  MoveL 1282 to (109.25, -79.9, 66.98) mm, rotated rx 117.25 ry 0 rz -126.43 deg; joints [128.975, -20.959, 32.859, -104.299, 40.472, 146.273, 25, -233.571]
  MoveL 1283 to (108.79, -81.97, 65.21) mm, rotated rx 116.26 ry 0 rz -127.74 deg; joints [128.667, -21.167, 33.266, -104.678, 40.231, 147.678, 25, -232.264]
  MoveL 1284 to (108.14, -83.32, 64.58) mm, rotated rx 116.26 ry 0 rz -127.74 deg; joints [128.686, -21.239, 33.332, -104.662, 40.248, 147.663, 25, -232.264]
  MoveL 1285 to (107.3, -84.35, 64.64) mm, rotated rx 116.25 ry 0 rz -127.85 deg; joints [128.711, -21.281, 33.364, -104.637, 40.269, 147.65, 25, -232.148]
  MoveL 1286 to (106.13, -85.42, 65.16) mm, rotated rx 116.5 ry 0 rz -129 deg; joints [128.756, -21.17, 33.217, -104.574, 40.301, 147.325, 25, -231.004]
  MoveL 1287 to (103.81, -89.56, 63.3) mm, rotated rx 115.13 ry 0 rz -131.76 deg; joints [128.34, -21.422, 33.746, -105.103, 39.98, 149.276, 25, -228.241]
  MoveL 1288 to (103.98, -91.37, 60.39) mm, rotated rx 113.92 ry 0 rz -132.27 deg; joints [127.986, -21.728, 34.311, -105.588, 39.715, 151.018, 25, -227.728]
  Set speed (16.7 mm/s)
  MoveL 1289 to (117.51, -103.67, 68.5) mm, rotated rx 113.92 ry 0 rz -132.27 deg; joints [127.572, -22.198, 34.1, -105.006, 39.145, 150.151, 25, -227.728]
  Set speed (1000.0 mm/s)
  MoveL 1290 to (138.84, -95.44, -29.33) mm, rotated rx 80.82 ry 0 rz -124.03 deg; joints [119.936, -25.445, 49.101, -124.867, 37.461, 205.459, 25, -235.972]
  Set speed (5.0 mm/s)
  MoveL 1291 to (122.47, -84.4, -26.14) mm, rotated rx 80.82 ry 0 rz -124.03 deg; joints [120.661, -24.792, 48.882, -124.547, 38.253, 205.426, 25, -235.972]
  Set speed (16.7 mm/s)
  MoveL 1292 to (121.83, -85.61, -25.22) mm, rotated rx 81.17 ry 0 rz -124.55 deg; joints [120.706, -24.83, 48.75, -124.321, 38.19, 204.807, 25, -235.447]
  MoveL 1293 to (121.51, -86.3, -24.42) mm, rotated rx 81.17 ry 0 rz -124.55 deg; joints [120.731, -24.874, 48.749, -124.248, 38.184, 204.727, 25, -235.447]
  MoveL 1294 to (121.4, -86.6, -23.9) mm, rotated rx 81.37 ry 0 rz -124.67 deg; joints [120.757, -24.895, 48.673, -124.119, 38.149, 204.372, 25, -235.327]
  MoveL 1295 to (121.32, -86.89, -23.19) mm, rotated rx 81.37 ry 0 rz -124.67 deg; joints [120.77, -24.915, 48.66, -124.07, 38.142, 204.317, 25, -235.327]
  MoveL 1296 to (121.66, -86.85, -21.5) mm, rotated rx 81.37 ry 0 rz -124.67 deg; joints [120.783, -24.917, 48.601, -123.991, 38.117, 204.223, 25, -235.327]
  MoveL 1297 to (123.29, -85.43, -17.57) mm, rotated rx 82.88 ry 0 rz -123.88 deg; joints [120.988, -25.05, 48.027, -123.022, 37.884, 201.596, 25, -236.124]
  MoveL 1298 to (123.63, -85.07, -16.92) mm, rotated rx 82.88 ry 0 rz -123.88 deg; joints [120.985, -25.03, 47.991, -123.009, 37.872, 201.577, 25, -236.124]
  MoveL 1299 to (124.64, -83.71, -16.25) mm, rotated rx 82.88 ry 0 rz -123.88 deg; joints [120.955, -24.952, 47.916, -123.043, 37.851, 201.606, 25, -236.124]
  MoveL 1300 to (124.99, -83.19, -16.24) mm, rotated rx 82.88 ry 0 rz -123.63 deg; joints [120.955, -24.952, 47.915, -123.042, 37.85, 201.602, 25, -236.366]
  MoveL 1301 to (125.61, -82.2, -16.51) mm, rotated rx 82.88 ry 0 rz -123.63 deg; joints [120.926, -24.894, 47.886, -123.104, 37.844, 201.666, 25, -236.366]
  MoveL 1302 to (128.29, -77.31, -19.31) mm, rotated rx 81.81 ry 0 rz -121.51 deg; joints [120.778, -24.803, 48.296, -123.794, 38.007, 203.536, 25, -238.495]
  MoveL 1303 to (128.77, -76.11, -20.82) mm, rotated rx 81.81 ry 0 rz -121.51 deg; joints [120.734, -24.729, 48.303, -123.926, 38.018, 203.681, 25, -238.495]
  MoveL 1304 to (128.6, -75.88, -22.52) mm, rotated rx 80.71 ry 0 rz -121.17 deg; joints [120.62, -24.664, 48.706, -124.541, 38.195, 205.508, 25, -238.828]
  MoveL 1305 to (129, -74.93, -23.4) mm, rotated rx 80.37 ry 0 rz -120.78 deg; joints [120.578, -24.627, 48.832, -124.756, 38.256, 206.097, 25, -239.222]
  MoveL 1306 to (129.03, -74.88, -23.37) mm, rotated rx 80.33 ry 0 rz -119.57 deg; joints [120.643, -24.776, 48.942, -124.646, 38.283, 206.031, 25, -240.434]
  MoveL 1307 to (130.64, -72.67, -21.45) mm, rotated rx 81.07 ry 0 rz -118.53 deg; joints [120.735, -24.856, 48.667, -124.175, 38.152, 204.743, 25, -241.473]
  MoveL 1308 to (131.06, -72.02, -21.04) mm, rotated rx 81.13 ry 0 rz -118.38 deg; joints [120.737, -24.845, 48.622, -124.138, 38.134, 204.631, 25, -241.615]
  MoveL 1309 to (133.41, -67.9, -19.93) mm, rotated rx 81.49 ry 0 rz -116.76 deg; joints [120.775, -24.857, 48.464, -123.919, 38.068, 204.011, 25, -243.236]
  MoveL 1310 to (133.8, -67.15, -19.89) mm, rotated rx 81.49 ry 0 rz -116.76 deg; joints [120.757, -24.816, 48.436, -123.951, 38.061, 204.043, 25, -243.236]
  MoveL 1311 to (134.25, -66.19, -20.09) mm, rotated rx 81.47 ry 0 rz -116.6 deg; joints [120.739, -24.783, 48.428, -123.998, 38.062, 204.113, 25, -243.403]
  MoveL 1312 to (135.7, -62.67, -21.57) mm, rotated rx 80.91 ry 0 rz -115.14 deg; joints [120.665, -24.726, 48.641, -124.361, 38.158, 205.101, 25, -244.859]
  MoveL 1313 to (137.15, -59.17, -22.28) mm, rotated rx 80.59 ry 0 rz -113.52 deg; joints [120.636, -24.714, 48.771, -124.54, 38.216, 205.634, 25, -246.485]
  MoveL 1314 to (137.34, -58.68, -22.4) mm, rotated rx 80.55 ry 0 rz -113.37 deg; joints [120.628, -24.703, 48.781, -124.57, 38.222, 205.704, 25, -246.63]
  MoveL 1315 to (138.52, -55.33, -23.62) mm, rotated rx 80.11 ry 0 rz -112.09 deg; joints [120.568, -24.642, 48.941, -124.865, 38.302, 206.49, 25, -247.906]
  MoveL 1316 to (138.88, -54.28, -23.91) mm, rotated rx 79.98 ry 0 rz -111.6 deg; joints [120.556, -24.635, 48.994, -124.94, 38.328, 206.712, 25, -248.398]
  MoveL 1317 to (141.71, -44.3, -27.64) mm, rotated rx 78.56 ry 0 rz -107.69 deg; joints [120.387, -24.444, 49.506, -125.843, 38.61, 209.189, 25, -252.307]
  MoveL 1318 to (141.88, -43.31, -28.3) mm, rotated rx 78.56 ry 0 rz -107.69 deg; joints [120.36, -24.387, 49.493, -125.918, 38.616, 209.27, 25, -252.307]
  MoveL 1319 to (141.91, -42.89, -28.8) mm, rotated rx 78.49 ry 0 rz -107.63 deg; joints [120.344, -24.361, 49.52, -125.988, 38.635, 209.422, 25, -252.372]
  MoveL 1320 to (141.9, -41.96, -30.15) mm, rotated rx 77.64 ry 0 rz -106.92 deg; joints [120.282, -24.295, 49.83, -126.436, 38.812, 210.814, 25, -253.083]
  MoveL 1321 to (142.62, -37.71, -32.31) mm, rotated rx 76.8 ry 0 rz -105.25 deg; joints [120.198, -24.163, 50.124, -126.951, 39.006, 212.263, 25, -254.745]
  MoveL 1322 to (142.69, -36.46, -33.43) mm, rotated rx 76.31 ry 0 rz -105.28 deg; joints [120.125, -24.017, 50.251, -127.3, 39.118, 213.17, 25, -254.72]
  MoveL 1323 to (142.55, -36.21, -34.26) mm, rotated rx 76.05 ry 0 rz -105.29 deg; joints [120.095, -23.958, 50.336, -127.474, 39.184, 213.632, 25, -254.707]
  MoveL 1324 to (141.72, -37.09, -36.6) mm, rotated rx 75.28 ry 0 rz -105.33 deg; joints [120.045, -23.861, 50.642, -127.92, 39.396, 214.954, 25, -254.667]
  MoveL 1325 to (141.78, -34.82, -38.6) mm, rotated rx 74.5 ry 0 rz -104.47 deg; joints [119.981, -23.71, 50.904, -128.385, 39.606, 216.3, 25, -255.53]
  MoveL 1326 to (141.86, -33.98, -39.09) mm, rotated rx 74.35 ry 0 rz -104.18 deg; joints [119.966, -23.674, 50.954, -128.484, 39.649, 216.57, 25, -255.818]
  MoveL 1327 to (141.57, -29.29, -43.66) mm, rotated rx 72.55 ry 0 rz -102.41 deg; joints [119.84, -23.287, 51.539, -129.529, 40.174, 219.654, 25, -257.589]
  MoveL 1328 to (141.21, -28.39, -45.4) mm, rotated rx 72.53 ry 0 rz -102.45 deg; joints [119.81, -23.204, 51.561, -129.658, 40.221, 219.826, 25, -257.553]
  MoveL 1329 to (140.47, -29.16, -47.19) mm, rotated rx 72.51 ry 0 rz -102.48 deg; joints [119.818, -23.207, 51.641, -129.72, 40.276, 219.933, 25, -257.518]
  MoveL 1330 to (139.72, -31.68, -47.77) mm, rotated rx 72.48 ry 0 rz -102.53 deg; joints [119.868, -23.318, 51.748, -129.659, 40.307, 219.911, 25, -257.472]
  MoveL 1331 to (139.19, -35.08, -46.94) mm, rotated rx 72.81 ry 0 rz -103.9 deg; joints [119.889, -23.395, 51.643, -129.47, 40.205, 219.343, 25, -256.101]
  MoveL 1332 to (139.1, -35.47, -46.89) mm, rotated rx 72.85 ry 0 rz -104.14 deg; joints [119.886, -23.392, 51.626, -129.46, 40.194, 219.294, 25, -255.858]
  MoveL 1333 to (138.15, -39.86, -46.17) mm, rotated rx 73.13 ry 0 rz -105.93 deg; joints [119.904, -23.456, 51.534, -129.296, 40.108, 218.805, 25, -254.07]
  MoveL 1334 to (137.98, -40.97, -45.71) mm, rotated rx 73.13 ry 0 rz -105.93 deg; joints [119.931, -23.521, 51.559, -129.229, 40.1, 218.733, 25, -254.07]
  MoveL 1335 to (137.95, -41.43, -45.38) mm, rotated rx 73.26 ry 0 rz -106.11 deg; joints [119.94, -23.551, 51.517, -129.153, 40.061, 218.507, 25, -253.89]
  MoveL 1336 to (137.95, -41.9, -44.95) mm, rotated rx 73.26 ry 0 rz -106.11 deg; joints [119.952, -23.582, 51.52, -129.113, 40.052, 218.463, 25, -253.89]
  MoveL 1337 to (138.12, -44.92, -41.35) mm, rotated rx 75.02 ry 0 rz -107.76 deg; joints [120.047, -23.866, 50.921, -128.179, 39.566, 215.545, 25, -252.236]
  MoveL 1338 to (137.32, -48.01, -40.54) mm, rotated rx 75.35 ry 0 rz -109.02 deg; joints [120.073, -23.928, 50.812, -127.987, 39.479, 214.989, 25, -250.98]
  MoveL 1339 to (137.34, -47.93, -40.55) mm, rotated rx 75.14 ry 0 rz -109.88 deg; joints [120.011, -23.783, 50.791, -128.175, 39.512, 215.397, 25, -250.12]
  MoveL 1340 to (135.25, -51.11, -43.62) mm, rotated rx 73.93 ry 0 rz -111.35 deg; joints [119.917, -23.537, 51.193, -128.891, 39.85, 217.485, 25, -248.653]
  MoveL 1341 to (134.45, -52.71, -44.19) mm, rotated rx 73.93 ry 0 rz -111.35 deg; joints [119.953, -23.617, 51.268, -128.846, 39.872, 217.449, 25, -248.653]
  MoveL 1342 to (134.28, -53.17, -44.17) mm, rotated rx 73.94 ry 0 rz -111.54 deg; joints [119.954, -23.619, 51.264, -128.84, 39.869, 217.429, 25, -248.459]
  MoveL 1343 to (133.34, -55.46, -44.11) mm, rotated rx 73.97 ry 0 rz -112.56 deg; joints [119.954, -23.619, 51.253, -128.83, 39.862, 217.393, 25, -247.435]
  MoveL 1344 to (132.43, -57.68, -44.06) mm, rotated rx 73.98 ry 0 rz -113.52 deg; joints [119.954, -23.623, 51.247, -128.819, 39.856, 217.36, 25, -246.485]
  MoveL 1345 to (132.15, -58.44, -43.91) mm, rotated rx 73.98 ry 0 rz -113.52 deg; joints [119.973, -23.667, 51.27, -128.779, 39.856, 217.319, 25, -246.485]
  MoveL 1346 to (131.99, -58.95, -43.73) mm, rotated rx 74.06 ry 0 rz -113.72 deg; joints [119.978, -23.682, 51.246, -128.736, 39.834, 217.192, 25, -246.275]
  MoveL 1347 to (131, -62.6, -41.54) mm, rotated rx 74.84 ry 0 rz -115.02 deg; joints [120.049, -23.868, 50.997, -128.247, 39.613, 215.819, 25, -244.982]
  MoveL 1348 to (128.38, -67.77, -41.64) mm, rotated rx 74.94 ry 0 rz -117.85 deg; joints [120.024, -23.813, 50.927, -128.26, 39.587, 215.717, 25, -242.151]
  Set speed (16.7 mm/s)
  MoveL 1349 to (145.45, -76.79, -46.84) mm, rotated rx 74.94 ry 0 rz -117.85 deg; joints [119.274, -24.456, 51.216, -128.772, 38.843, 215.939, 25, -242.151]
  Set speed (1000.0 mm/s)
  MoveL 1350 to (145.71, -79, -42.14) mm, rotated rx 75.13 ry 0 rz -117.87 deg; joints [119.357, -24.65, 51.093, -128.369, 38.703, 215.283, 25, -242.133]
  Set speed (5.0 mm/s)
  MoveL 1351 to (128.62, -69.96, -37.01) mm, rotated rx 75.13 ry 0 rz -117.87 deg; joints [120.107, -24.006, 50.807, -127.869, 39.451, 215.072, 25, -242.133]
  Set speed (16.7 mm/s)
  MoveL 1352 to (129.85, -68.52, -35.3) mm, rotated rx 75.8 ry 0 rz -117.14 deg; joints [120.165, -24.128, 50.579, -127.467, 39.279, 213.919, 25, -242.855]
  MoveL 1353 to (129.85, -68.52, -35.32) mm, rotated rx 76.99 ry 0 rz -117 deg; joints [120.26, -24.308, 50.268, -126.882, 39.05, 212.028, 25, -243.001]
  MoveL 1354 to (129.74, -69.29, -34.22) mm, rotated rx 77.8 ry 0 rz -117.78 deg; joints [120.303, -24.361, 49.969, -126.485, 38.871, 210.73, 25, -242.216]
  MoveL 1355 to (129.04, -70.88, -33.63) mm, rotated rx 78.03 ry 0 rz -118.46 deg; joints [120.327, -24.396, 49.888, -126.342, 38.819, 210.329, 25, -241.541]
  MoveL 1356 to (128.8, -71.45, -33.34) mm, rotated rx 78.08 ry 0 rz -118.56 deg; joints [120.341, -24.424, 49.876, -126.287, 38.806, 210.213, 25, -241.44]
  MoveL 1357 to (128.09, -73.34, -31.98) mm, rotated rx 78.67 ry 0 rz -119.48 deg; joints [120.394, -24.489, 49.659, -125.945, 38.679, 209.218, 25, -240.525]
  MoveL 1358 to (127.59, -74.37, -31.59) mm, rotated rx 78.82 ry 0 rz -119.92 deg; joints [120.411, -24.511, 49.604, -125.85, 38.646, 208.953, 25, -240.079]
  MoveL 1359 to (123.08, -82.67, -28.71) mm, rotated rx 79.95 ry 0 rz -123.6 deg; joints [120.537, -24.655, 49.192, -125.145, 38.416, 206.991, 25, -236.396]
  Set speed (16.7 mm/s)
  MoveL 1360 to (139.48, -93.57, -32.2) mm, rotated rx 79.95 ry 0 rz -123.6 deg; joints [119.808, -25.307, 49.422, -125.495, 37.63, 207.055, 25, -236.396]
  Set speed (1000.0 mm/s)
  MoveL 1361 to (86.56, -126.27, -76.23) mm, rotated rx 62.7 ry 0 rz -145.47 deg; joints [118.894, -20.973, 54.737, -135.201, 43.294, 236.447, 25, -214.527]
  Set speed (5.0 mm/s)
  MoveL 1362 to (76.48, -111.63, -67.06) mm, rotated rx 62.7 ry 0 rz -145.47 deg; joints [119.661, -20.42, 54.326, -134.408, 43.847, 235.941, 25, -214.527]
  Set speed (16.7 mm/s)
  MoveL 1363 to (78.17, -110.46, -67.04) mm, rotated rx 62.7 ry 0 rz -144.73 deg; joints [119.655, -20.405, 54.316, -134.418, 43.845, 235.95, 25, -215.272]
  MoveL 1364 to (82.31, -108.27, -65.64) mm, rotated rx 63.33 ry 0 rz -142.43 deg; joints [119.663, -20.682, 54.196, -134.111, 43.574, 234.894, 25, -217.574]
  MoveL 1365 to (83.1, -107.77, -65.47) mm, rotated rx 63.37 ry 0 rz -142.18 deg; joints [119.655, -20.681, 54.173, -134.104, 43.553, 234.839, 25, -217.817]
  MoveL 1366 to (86.56, -105.46, -64.75) mm, rotated rx 63.68 ry 0 rz -140.42 deg; joints [119.653, -20.796, 54.1, -133.964, 43.422, 234.337, 25, -219.58]
  MoveL 1367 to (90.08, -104.34, -61.68) mm, rotated rx 65.21 ry 0 rz -138.47 deg; joints [119.676, -21.383, 53.775, -133.232, 42.807, 231.82, 25, -221.529]
  MoveL 1368 to (92.29, -104.07, -58.82) mm, rotated rx 66.58 ry 0 rz -137.55 deg; joints [119.696, -21.844, 53.439, -132.573, 42.276, 229.569, 25, -222.448]
  MoveL 1369 to (93.65, -103.42, -57.81) mm, rotated rx 66.58 ry 0 rz -137.55 deg; joints [119.665, -21.799, 53.365, -132.585, 42.238, 229.563, 25, -222.448]
  MoveL 1370 to (94.29, -102.92, -57.66) mm, rotated rx 66.61 ry 0 rz -137.46 deg; joints [119.653, -21.778, 53.336, -132.592, 42.225, 229.541, 25, -222.535]
  MoveL 1371 to (95.59, -101.74, -57.6) mm, rotated rx 66.63 ry 0 rz -136.74 deg; joints [119.653, -21.786, 53.329, -132.579, 42.214, 229.497, 25, -223.256]
  MoveL 1372 to (97.07, -100.77, -56.82) mm, rotated rx 67.03 ry 0 rz -135.66 deg; joints [119.68, -21.954, 53.256, -132.353, 42.069, 228.812, 25, -224.345]
  MoveL 1373 to (99.36, -99.94, -54.29) mm, rotated rx 68.34 ry 0 rz -134.37 deg; joints [119.729, -22.38, 52.94, -131.68, 41.604, 226.634, 25, -225.629]
  MoveL 1374 to (99.89, -99.67, -53.81) mm, rotated rx 68.34 ry 0 rz -134.37 deg; joints [119.718, -22.364, 52.909, -131.68, 41.587, 226.627, 25, -225.629]
  MoveL 1375 to (100.33, -99.39, -53.5) mm, rotated rx 68.42 ry 0 rz -134.25 deg; joints [119.716, -22.378, 52.877, -131.644, 41.555, 226.502, 25, -225.75]
  MoveL 1376 to (103.28, -97.29, -51.72) mm, rotated rx 69.14 ry 0 rz -132.81 deg; joints [119.74, -22.584, 52.669, -131.265, 41.295, 225.29, 25, -227.188]
  MoveL 1377 to (103.68, -96.97, -51.52) mm, rotated rx 69.17 ry 0 rz -132.72 deg; joints [119.735, -22.582, 52.647, -131.252, 41.279, 225.238, 25, -227.281]
  MoveL 1378 to (105.78, -94.99, -50.95) mm, rotated rx 69.35 ry 0 rz -131.73 deg; joints [119.733, -22.613, 52.576, -131.168, 41.211, 224.943, 25, -228.269]
  MoveL 1379 to (106.4, -94.3, -50.95) mm, rotated rx 69.35 ry 0 rz -131.73 deg; joints [119.713, -22.566, 52.545, -131.205, 41.208, 224.978, 25, -228.269]
  MoveL 1380 to (106.81, -93.76, -51.06) mm, rotated rx 69.31 ry 0 rz -131.46 deg; joints [119.711, -22.553, 52.558, -131.229, 41.224, 225.056, 25, -228.542]
  MoveL 1381 to (109.17, -90.01, -52.73) mm, rotated rx 68.69 ry 0 rz -129.9 deg; joints [119.679, -22.348, 52.723, -131.582, 41.448, 226.121, 25, -230.098]
  MoveL 1382 to (109.1, -90.07, -52.8) mm, rotated rx 68.9 ry 0 rz -128.78 deg; joints [119.745, -22.541, 52.773, -131.384, 41.397, 225.686, 25, -231.217]
  MoveL 1383 to (110.45, -89.31, -51.3) mm, rotated rx 69.51 ry 0 rz -128.21 deg; joints [119.767, -22.71, 52.596, -131.062, 41.182, 224.665, 25, -231.793]
  MoveL 1384 to (110.71, -89.18, -50.98) mm, rotated rx 69.68 ry 0 rz -128.06 deg; joints [119.775, -22.758, 52.551, -130.973, 41.126, 224.384, 25, -231.935]
  MoveL 1385 to (114.23, -86.61, -47.5) mm, rotated rx 70.95 ry 0 rz -126.52 deg; joints [119.826, -23.082, 52.15, -130.28, 40.688, 222.23, 25, -233.485]
  MoveL 1386 to (115.16, -85.68, -46.95) mm, rotated rx 70.95 ry 0 rz -126.52 deg; joints [119.8, -23.028, 52.092, -130.305, 40.668, 222.248, 25, -233.485]
  MoveL 1387 to (115.49, -85.28, -46.88) mm, rotated rx 70.98 ry 0 rz -126.31 deg; joints [119.801, -23.035, 52.084, -130.291, 40.659, 222.203, 25, -233.692]
  MoveL 1388 to (116.72, -83.72, -46.58) mm, rotated rx 71.09 ry 0 rz -125.5 deg; joints [119.809, -23.067, 52.048, -130.222, 40.621, 221.998, 25, -234.503]
  MoveL 1389 to (117.65, -83.33, -44.95) mm, rotated rx 71.52 ry 0 rz -125.1 deg; joints [119.837, -23.19, 51.907, -129.953, 40.469, 221.236, 25, -234.901]
  MoveL 1390 to (118.89, -81.86, -44.41) mm, rotated rx 71.96 ry 0 rz -124.69 deg; joints [119.84, -23.24, 51.754, -129.767, 40.342, 220.553, 25, -235.312]
  MoveL 1391 to (119.23, -81.32, -44.49) mm, rotated rx 71.93 ry 0 rz -124.44 deg; joints [119.838, -23.232, 51.765, -129.786, 40.352, 220.611, 25, -235.565]
  MoveL 1392 to (122.81, -74.48, -46.64) mm, rotated rx 71.1 ry 0 rz -121.52 deg; joints [119.785, -23.01, 52.011, -130.267, 40.617, 222.036, 25, -238.477]
  MoveL 1393 to (123.08, -74.04, -46.65) mm, rotated rx 71.07 ry 0 rz -121.16 deg; joints [119.791, -23.024, 52.032, -130.267, 40.627, 222.073, 25, -238.838]
  MoveL 1394 to (125.13, -70.14, -47.21) mm, rotated rx 70.84 ry 0 rz -119.41 deg; joints [119.78, -22.967, 52.101, -130.391, 40.701, 222.454, 25, -240.594]
  MoveL 1395 to (125.67, -68.6, -48.04) mm, rotated rx 70.81 ry 0 rz -119.41 deg; joints [119.74, -22.86, 52.077, -130.509, 40.727, 222.618, 25, -240.594]
  MoveL 1396 to (125.64, -67.91, -49.09) mm, rotated rx 70.78 ry 0 rz -119.41 deg; joints [119.723, -22.803, 52.09, -130.592, 40.762, 222.739, 25, -240.594]
  MoveL 1397 to (124.81, -67.96, -51.11) mm, rotated rx 70.74 ry 0 rz -119.41 deg; joints [119.722, -22.772, 52.168, -130.687, 40.832, 222.907, 25, -240.594]
  MoveL 1398 to (123.74, -68.7, -52.68) mm, rotated rx 69.66 ry 0 rz -120.05 deg; joints [119.672, -22.487, 52.448, -131.236, 41.17, 224.686, 25, -239.954]
  MoveL 1399 to (123.37, -68.58, -53.7) mm, rotated rx 69.24 ry 0 rz -120.08 deg; joints [119.657, -22.372, 52.569, -131.456, 41.316, 225.382, 25, -239.918]
  MoveL 1400 to (122.17, -69.3, -55.43) mm, rotated rx 67.67 ry 0 rz -120.12 deg; joints [119.641, -22.022, 53.002, -132.132, 41.828, 227.851, 25, -239.877]
  MoveL 1401 to (122.63, -67.73, -56.41) mm, rotated rx 67.27 ry 0 rz -119.48 deg; joints [119.632, -21.902, 53.112, -132.333, 41.977, 228.509, 25, -240.525]
  MoveL 1402 to (123.25, -65.21, -58) mm, rotated rx 66.64 ry 0 rz -118.48 deg; joints [119.619, -21.697, 53.284, -132.654, 42.223, 229.568, 25, -241.524]
  MoveL 1403 to (123.68, -64.08, -58.35) mm, rotated rx 66.37 ry 0 rz -117.71 deg; joints [119.63, -21.654, 53.371, -132.748, 42.318, 229.971, 25, -242.288]
  MoveL 1404 to (123.84, -63.54, -58.59) mm, rotated rx 66.37 ry 0 rz -117.71 deg; joints [119.618, -21.618, 53.358, -132.78, 42.326, 230.006, 25, -242.288]
  MoveL 1405 to (124.29, -61.65, -59.63) mm, rotated rx 65.93 ry 0 rz -116.91 deg; joints [119.615, -21.478, 53.476, -132.991, 42.5, 230.731, 25, -243.086]
  MoveL 1406 to (124.3, -61.62, -59.61) mm, rotated rx 66.05 ry 0 rz -115.66 deg; joints [119.681, -21.662, 53.553, -132.829, 42.468, 230.435, 25, -244.336]
  MoveL 1407 to (126.02, -59.94, -57.71) mm, rotated rx 66.83 ry 0 rz -114.74 deg; joints [119.691, -21.914, 53.344, -132.444, 42.161, 229.141, 25, -245.256]
  MoveL 1408 to (128.44, -59.64, -52.46) mm, rotated rx 69.46 ry 0 rz -113.92 deg; joints [119.774, -22.7, 52.656, -131.115, 41.233, 224.793, 25, -246.078]
  MoveL 1409 to (128.8, -59.51, -51.74) mm, rotated rx 69.54 ry 0 rz -113.9 deg; joints [119.774, -22.725, 52.613, -131.056, 41.188, 224.634, 25, -246.103]
  MoveL 1410 to (129.78, -58.91, -49.96) mm, rotated rx 70.26 ry 0 rz -113.52 deg; joints [119.804, -22.918, 52.399, -130.669, 40.941, 223.421, 25, -246.485]
  MoveL 1411 to (130.23, -58.65, -49.07) mm, rotated rx 70.48 ry 0 rz -113.43 deg; joints [119.81, -22.974, 52.315, -130.539, 40.855, 223.029, 25, -246.565]
  MoveL 1412 to (132.89, -56.13, -44.69) mm, rotated rx 72.23 ry 0 rz -112.09 deg; joints [119.903, -23.404, 51.775, -129.566, 40.293, 220.062, 25, -247.906]
  MoveL 1413 to (133.87, -54.54, -43.72) mm, rotated rx 72.23 ry 0 rz -112.09 deg; joints [119.868, -23.33, 51.687, -129.594, 40.26, 220.077, 25, -247.906]
  MoveL 1414 to (134.4, -52.63, -44.42) mm, rotated rx 72.23 ry 0 rz -112.09 deg; joints [119.821, -23.216, 51.64, -129.707, 40.272, 220.196, 25, -247.906]
  MoveL 1415 to (134.45, -52.04, -44.98) mm, rotated rx 72.01 ry 0 rz -111.87 deg; joints [119.808, -23.164, 51.71, -129.832, 40.34, 220.572, 25, -248.133]
  MoveL 1416 to (134.35, -51.3, -46.09) mm, rotated rx 72.01 ry 0 rz -111.87 deg; joints [119.789, -23.109, 51.718, -129.911, 40.367, 220.663, 25, -248.133]
  MoveL 1417 to (132.92, -49.01, -52.29) mm, rotated rx 68.94 ry 0 rz -110.79 deg; joints [119.678, -22.397, 52.641, -131.472, 41.36, 225.719, 25, -249.211]
  MoveL 1418 to (133.31, -45.82, -54.18) mm, rotated rx 68.18 ry 0 rz -109.52 deg; joints [119.654, -22.176, 52.86, -131.871, 41.638, 227, 25, -250.479]
  MoveL 1419 to (133.02, -44.52, -55.95) mm, rotated rx 68.18 ry 0 rz -109.52 deg; joints [119.625, -22.073, 52.864, -131.994, 41.691, 227.145, 25, -250.479]
  MoveL 1420 to (132.73, -44.42, -56.71) mm, rotated rx 68.1 ry 0 rz -109.51 deg; joints [119.623, -22.035, 52.902, -132.059, 41.739, 227.309, 25, -250.485]
  MoveL 1421 to (132.12, -44.47, -58.08) mm, rotated rx 67.54 ry 0 rz -109.62 deg; joints [119.61, -21.865, 53.057, -132.344, 41.95, 228.243, 25, -250.382]
  MoveL 1422 to (131.58, -43.17, -60.26) mm, rotated rx 66.1 ry 0 rz -109.11 deg; joints [119.593, -21.453, 53.419, -132.99, 42.465, 230.539, 25, -250.887]
  MoveL 1423 to (131.38, -42.9, -60.88) mm, rotated rx 66.1 ry 0 rz -109.11 deg; joints [119.589, -21.426, 53.427, -133.024, 42.486, 230.582, 25, -250.887]
  MoveL 1424 to (131.19, -42.76, -61.38) mm, rotated rx 65.89 ry 0 rz -109.08 deg; joints [119.587, -21.356, 53.482, -133.125, 42.57, 230.927, 25, -250.916]
  MoveL 1425 to (130.01, -41.88, -64.4) mm, rotated rx 64.63 ry 0 rz -108.89 deg; joints [119.585, -20.922, 53.806, -133.721, 43.089, 233.006, 25, -251.105]
  MoveL 1426 to (130.03, -41.89, -64.35) mm, rotated rx 63.97 ry 0 rz -108.41 deg; joints [119.612, -20.8, 53.972, -133.912, 43.306, 233.942, 25, -251.586]
  MoveL 1427 to (130.19, -37.44, -66.76) mm, rotated rx 62.96 ry 0 rz -106.61 deg; joints [119.623, -20.427, 54.215, -134.364, 43.741, 235.586, 25, -253.393]
  MoveL 1428 to (129.62, -36.05, -68.6) mm, rotated rx 62.96 ry 0 rz -106.61 deg; joints [119.6, -20.305, 54.213, -134.48, 43.812, 235.73, 25, -253.393]
  MoveL 1429 to (129.03, -35.2, -70.14) mm, rotated rx 62.01 ry 0 rz -106.27 deg; joints [119.622, -19.968, 54.423, -134.857, 44.208, 237.227, 25, -253.73]
  MoveL 1430 to (128.75, -34.95, -70.79) mm, rotated rx 61.95 ry 0 rz -106.25 deg; joints [119.621, -19.922, 54.44, -134.904, 44.253, 237.343, 25, -253.745]
  MoveL 1431 to (128.62, -34.84, -71.06) mm, rotated rx 61.16 ry 0 rz -105.78 deg; joints [119.661, -19.714, 54.62, -135.137, 44.551, 238.497, 25, -254.216]
  MoveL 1432 to (128.52, -33.37, -71.94) mm, rotated rx 60.78 ry 0 rz -105.19 deg; joints [119.673, -19.561, 54.702, -135.291, 44.724, 239.1, 25, -254.815]
  MoveL 1433 to (128.3, -32.51, -72.73) mm, rotated rx 60.78 ry 0 rz -105.19 deg; joints [119.659, -19.492, 54.69, -135.348, 44.757, 239.169, 25, -254.815]
  MoveL 1434 to (128.05, -32.17, -73.32) mm, rotated rx 60.73 ry 0 rz -105.16 deg; joints [119.658, -19.444, 54.703, -135.392, 44.799, 239.279, 25, -254.842]
  MoveL 1435 to (127.47, -31.67, -74.53) mm, rotated rx 60.2 ry 0 rz -105.01 deg; joints [119.677, -19.224, 54.813, -135.601, 45.045, 240.117, 25, -254.986]
  MoveL 1436 to (126.85, -29.7, -76.38) mm, rotated rx 59.02 ry 0 rz -104.04 deg; joints [119.736, -18.777, 55.051, -136.007, 45.57, 241.925, 25, -255.964]
  MoveL 1437 to (126.72, -29.34, -76.74) mm, rotated rx 58.91 ry 0 rz -103.94 deg; joints [119.739, -18.719, 55.072, -136.056, 45.629, 242.109, 25, -256.061]
  MoveL 1438 to (125.84, -27.3, -78.9) mm, rotated rx 57.96 ry 0 rz -103.16 deg; joints [119.79, -18.293, 55.252, -136.404, 46.094, 243.607, 25, -256.844]
  MoveL 1439 to (125.36, -26.75, -79.85) mm, rotated rx 57.96 ry 0 rz -103.16 deg; joints [119.786, -18.231, 55.253, -136.451, 46.138, 243.671, 25, -256.844]
  MoveL 1440 to (124.53, -26.64, -81.17) mm, rotated rx 57.8 ry 0 rz -103.13 deg; joints [119.803, -18.124, 55.302, -136.534, 46.26, 243.96, 25, -256.867]
  MoveL 1441 to (122.66, -27.32, -83.76) mm, rotated rx 56.63 ry 0 rz -103.63 deg; joints [119.878, -17.577, 55.507, -136.935, 46.848, 245.785, 25, -256.371]
  MoveL 1442 to (120.31, -27.21, -87.13) mm, rotated rx 54.87 ry 0 rz -103.9 deg; joints [120.005, -16.737, 55.773, -137.482, 47.728, 248.466, 25, -256.103]
  MoveL 1443 to (119.84, -27.31, -87.74) mm, rotated rx 54.87 ry 0 rz -103.9 deg; joints [120.014, -16.718, 55.79, -137.494, 47.759, 248.492, 25, -256.103]
  MoveL 1444 to (119.51, -27.47, -88.15) mm, rotated rx 54.68 ry 0 rz -104.01 deg; joints [120.03, -16.622, 55.818, -137.551, 47.859, 248.784, 25, -255.994]
  MoveL 1445 to (115.59, -30.1, -92.42) mm, rotated rx 52.79 ry 0 rz -105.59 deg; joints [120.21, -15.647, 56.084, -138.086, 48.872, 251.646, 25, -254.408]
  MoveL 1446 to (115.26, -30.28, -92.76) mm, rotated rx 52.59 ry 0 rz -105.75 deg; joints [120.229, -15.542, 56.106, -138.139, 48.976, 251.946, 25, -254.253]
  MoveL 1447 to (111.45, -33.08, -96.4) mm, rotated rx 50.93 ry 0 rz -107.49 deg; joints [120.414, -14.64, 56.303, -138.554, 49.89, 254.433, 25, -252.511]
  MoveL 1448 to (110.88, -33.62, -96.87) mm, rotated rx 50.85 ry 0 rz -107.62 deg; joints [120.435, -14.599, 56.33, -138.566, 49.951, 254.553, 25, -252.381]
  MoveL 1449 to (109.03, -35.76, -98.19) mm, rotated rx 50.24 ry 0 rz -108.84 deg; joints [120.512, -14.258, 56.397, -138.705, 50.295, 255.465, 25, -251.157]
  MoveL 1450 to (105.97, -37.85, -100.72) mm, rotated rx 48.8 ry 0 rz -110.6 deg; joints [120.676, -13.436, 56.5, -139.018, 51.071, 257.572, 25, -249.397]
  MoveL 1451 to (105.56, -38.13, -101.04) mm, rotated rx 48.65 ry 0 rz -110.79 deg; joints [120.697, -13.35, 56.513, -139.047, 51.156, 257.79, 25, -249.211]
  MoveL 1452 to (102.4, -40.39, -103.39) mm, rotated rx 47.47 ry 0 rz -112.43 deg; joints [120.859, -12.658, 56.599, -139.269, 51.821, 259.506, 25, -247.568]
  MoveL 1453 to (101.99, -40.57, -103.73) mm, rotated rx 47.27 ry 0 rz -112.63 deg; joints [120.885, -12.539, 56.609, -139.306, 51.931, 259.796, 25, -247.369]
  MoveL 1454 to (97.91, -42.95, -106.66) mm, rotated rx 45.71 ry 0 rz -114.67 deg; joints [121.112, -11.601, 56.688, -139.562, 52.809, 262.032, 25, -245.333]
  MoveL 1455 to (96.76, -44.15, -107.22) mm, rotated rx 45.71 ry 0 rz -114.67 deg; joints [121.157, -11.635, 56.749, -139.525, 52.849, 262.024, 25, -245.333]
  MoveL 1456 to (95.06, -46.9, -107.57) mm, rotated rx 45.52 ry 0 rz -116.47 deg; joints [121.184, -11.51, 56.751, -139.558, 52.959, 262.305, 25, -243.531]
  MoveL 1457 to (92.2, -49.19, -109.03) mm, rotated rx 44.59 ry 0 rz -118.79 deg; joints [121.304, -10.915, 56.748, -139.711, 53.465, 263.628, 25, -241.206]
  MoveL 1458 to (91.24, -50.42, -109.28) mm, rotated rx 44.59 ry 0 rz -118.79 deg; joints [121.343, -10.968, 56.806, -139.67, 53.486, 263.606, 25, -241.206]
  MoveL 1459 to (90.83, -51.64, -109.04) mm, rotated rx 44.6 ry 0 rz -118.95 deg; joints [121.359, -11.035, 56.841, -139.636, 53.469, 263.559, 25, -241.05]
  MoveL 1460 to (90.6, -53.29, -108.43) mm, rotated rx 44.94 ry 0 rz -119.8 deg; joints [121.306, -11.241, 56.831, -139.591, 53.28, 263.086, 25, -240.198]
  MoveL 1461 to (90.59, -53.38, -108.39) mm, rotated rx 45.04 ry 0 rz -120.88 deg; joints [121.25, -11.208, 56.757, -139.634, 53.224, 262.985, 25, -239.119]
  MoveL 1462 to (89.12, -54.97, -108.83) mm, rotated rx 44.81 ry 0 rz -122.05 deg; joints [121.287, -11.062, 56.765, -139.667, 53.358, 263.32, 25, -237.955]
  MoveL 1463 to (88.6, -55.68, -108.89) mm, rotated rx 44.81 ry 0 rz -122.05 deg; joints [121.307, -11.098, 56.797, -139.642, 53.365, 263.304, 25, -237.955]
  MoveL 1464 to (88.21, -56.59, -108.74) mm, rotated rx 44.81 ry 0 rz -122.14 deg; joints [121.323, -11.148, 56.827, -139.616, 53.355, 263.272, 25, -237.862]
  MoveL 1465 to (87.77, -58.17, -108.26) mm, rotated rx 45.07 ry 0 rz -122.99 deg; joints [121.281, -11.31, 56.819, -139.579, 53.207, 262.9, 25, -237.008]
  MoveL 1466 to (87.47, -59.22, -107.93) mm, rotated rx 45.14 ry 0 rz -123.28 deg; joints [121.279, -11.389, 56.834, -139.551, 53.157, 262.785, 25, -236.716]
  MoveL 1467 to (87.01, -63.11, -106.08) mm, rotated rx 46.14 ry 0 rz -125.16 deg; joints [121.126, -12, 56.793, -139.401, 52.592, 261.358, 25, -234.841]
  MoveL 1468 to (87.5, -64.69, -104.72) mm, rotated rx 46.14 ry 0 rz -125.16 deg; joints [121.126, -12.14, 56.823, -139.346, 52.508, 261.267, 25, -234.841]
  MoveL 1469 to (88.16, -65.07, -103.92) mm, rotated rx 46.27 ry 0 rz -125.17 deg; joints [121.096, -12.252, 56.81, -139.317, 52.4, 261.057, 25, -234.833]
  MoveL 1470 to (89.29, -65.35, -102.77) mm, rotated rx 46.86 ry 0 rz -124.95 deg; joints [121.009, -12.61, 56.777, -139.216, 52.063, 260.197, 25, -235.05]
  MoveL 1471 to (89.25, -65.37, -102.8) mm, rotated rx 47.65 ry 0 rz -125.17 deg; joints [120.914, -12.96, 56.725, -139.117, 51.714, 259.139, 25, -234.827]
  MoveL 1472 to (89.38, -66.4, -102.03) mm, rotated rx 48.05 ry 0 rz -125.57 deg; joints [120.858, -13.197, 56.698, -139.042, 51.488, 258.554, 25, -234.433]
  MoveL 1473 to (90.2, -67.77, -100.38) mm, rotated rx 49.14 ry 0 rz -127.6 deg; joints [120.649, -13.634, 56.495, -138.941, 50.904, 257.082, 25, -232.402]
  MoveL 1474 to (88.7, -68.61, -101.15) mm, rotated rx 48.75 ry 0 rz -128.41 deg; joints [120.699, -13.41, 56.526, -139.02, 51.121, 257.652, 25, -231.591]
  MoveL 1475 to (87.69, -69.33, -101.54) mm, rotated rx 48.76 ry 0 rz -128.44 deg; joints [120.728, -13.445, 56.57, -138.992, 51.142, 257.626, 25, -231.559]
  MoveL 1476 to (86.89, -70.89, -101.15) mm, rotated rx 48.78 ry 0 rz -128.48 deg; joints [120.757, -13.555, 56.626, -138.93, 51.115, 257.543, 25, -231.515]
  MoveL 1477 to (87.23, -72.68, -99.58) mm, rotated rx 48.8 ry 0 rz -128.54 deg; joints [120.757, -13.715, 56.651, -138.859, 51.013, 257.407, 25, -231.457]
  MoveL 1478 to (88.09, -73.52, -98.19) mm, rotated rx 49.5 ry 0 rz -128.6 deg; joints [120.669, -14.115, 56.592, -138.712, 50.625, 256.382, 25, -231.4]
  MoveL 1479 to (88.4, -75.8, -96.15) mm, rotated rx 51.34 ry 0 rz -130.18 deg; joints [120.436, -14.969, 56.369, -138.38, 49.704, 253.776, 25, -229.819]
  MoveL 1480 to (86.63, -79.11, -95.09) mm, rotated rx 51.86 ry 0 rz -131.98 deg; joints [120.379, -15.252, 56.312, -138.252, 49.421, 253, 25, -228.023]
  MoveL 1481 to (86.26, -79.54, -95.08) mm, rotated rx 51.93 ry 0 rz -132.56 deg; joints [120.36, -15.249, 56.283, -138.26, 49.392, 252.929, 25, -227.437]
  MoveL 1482 to (79.34, -84.7, -96.64) mm, rotated rx 51.14 ry 0 rz -137.15 deg; joints [120.428, -14.785, 56.339, -138.476, 49.815, 254.117, 25, -222.853]
  MoveL 1483 to (78.82, -85.12, -96.69) mm, rotated rx 51.14 ry 0 rz -137.28 deg; joints [120.438, -14.799, 56.355, -138.466, 49.822, 254.117, 25, -222.725]
  MoveL 1484 to (77.12, -86.67, -96.68) mm, rotated rx 51.14 ry 0 rz -138.33 deg; joints [120.441, -14.81, 56.361, -138.459, 49.819, 254.105, 25, -221.674]
  MoveL 1485 to (76.85, -86.83, -96.76) mm, rotated rx 51.08 ry 0 rz -138.77 deg; joints [120.435, -14.751, 56.345, -138.491, 49.848, 254.209, 25, -221.231]
  MoveL 1486 to (70.66, -88.85, -99.6) mm, rotated rx 49.55 ry 0 rz -142.16 deg; joints [120.598, -13.869, 56.463, -138.854, 50.679, 256.482, 25, -217.843]
  MoveL 1487 to (69.62, -89.36, -99.87) mm, rotated rx 49.55 ry 0 rz -142.16 deg; joints [120.627, -13.907, 56.507, -138.825, 50.697, 256.467, 25, -217.843]
  MoveL 1488 to (68.94, -89.84, -99.91) mm, rotated rx 49.53 ry 0 rz -142.58 deg; joints [120.629, -13.896, 56.509, -138.83, 50.709, 256.497, 25, -217.423]
  MoveL 1489 to (62.76, -94.08, -100.08) mm, rotated rx 49.44 ry 0 rz -146.33 deg; joints [120.642, -13.851, 56.519, -138.845, 50.756, 256.62, 25, -213.673]
  MoveL 1490 to (62.53, -94.11, -100.2) mm, rotated rx 49.32 ry 0 rz -146.84 deg; joints [120.638, -13.753, 56.499, -138.891, 50.813, 256.806, 25, -213.163]
  MoveL 1491 to (54.8, -96.96, -101.99) mm, rotated rx 48.43 ry 0 rz -150.89 deg; joints [120.758, -13.241, 56.575, -139.068, 51.314, 258.112, 25, -209.111]
  MoveL 1492 to (52.96, -98.33, -101.65) mm, rotated rx 48.43 ry 0 rz -150.89 deg; joints [120.803, -13.372, 56.657, -138.991, 51.299, 258.039, 25, -209.111]
  MoveL 1493 to (52.64, -98.87, -101.3) mm, rotated rx 48.51 ry 0 rz -151.03 deg; joints [120.796, -13.445, 56.659, -138.962, 51.241, 257.899, 25, -208.971]
  MoveL 1494 to (51.49, -101.18, -99.59) mm, rotated rx 49.39 ry 0 rz -152.11 deg; joints [120.683, -13.948, 56.588, -138.784, 50.755, 256.621, 25, -207.891]
  MoveL 1495 to (51.53, -102.66, -98.05) mm, rotated rx 49.39 ry 0 rz -152.11 deg; joints [120.677, -14.073, 56.598, -138.728, 50.665, 256.527, 25, -207.891]
  MoveL 1496 to (52.62, -103.3, -96.79) mm, rotated rx 49.5 ry 0 rz -152.09 deg; joints [120.635, -14.172, 56.555, -138.699, 50.538, 256.318, 25, -207.912]
  MoveL 1497 to (54.87, -103.58, -95.22) mm, rotated rx 50.27 ry 0 rz -151.18 deg; joints [120.543, -14.602, 56.482, -138.527, 50.116, 255.189, 25, -208.816]
  MoveL 1498 to (56.61, -104.63, -93.02) mm, rotated rx 52.15 ry 0 rz -150.4 deg; joints [120.369, -15.565, 56.319, -138.089, 49.188, 252.456, 25, -209.597]
  MoveL 1499 to (56.93, -106.13, -91.13) mm, rotated rx 53.06 ry 0 rz -150.62 deg; joints [120.277, -16.049, 56.206, -137.846, 48.698, 251.082, 25, -209.379]
  MoveL 1500 to (57.12, -106.52, -90.54) mm, rotated rx 53.06 ry 0 rz -150.62 deg; joints [120.272, -16.082, 56.2, -137.829, 48.666, 251.051, 25, -209.379]
  MoveL 1501 to (57.34, -106.77, -90.11) mm, rotated rx 53.16 ry 0 rz -150.61 deg; joints [120.259, -16.146, 56.182, -137.795, 48.599, 250.883, 25, -209.393]
  MoveL 1502 to (58.34, -107.62, -88.43) mm, rotated rx 53.95 ry 0 rz -150.4 deg; joints [120.186, -16.552, 56.075, -137.571, 48.182, 249.689, 25, -209.604]
  MoveL 1503 to (58.38, -109.47, -86.11) mm, rotated rx 55.51 ry 0 rz -150.83 deg; joints [120.063, -17.279, 55.858, -137.132, 47.423, 247.362, 25, -209.175]
  MoveL 1504 to (58.45, -109.83, -85.61) mm, rotated rx 55.56 ry 0 rz -150.83 deg; joints [120.058, -17.33, 55.847, -137.1, 47.375, 247.254, 25, -209.168]
  MoveL 1505 to (58.95, -110.73, -84.09) mm, rotated rx 56.15 ry 0 rz -150.83 deg; joints [120.013, -17.625, 55.75, -136.904, 47.063, 246.34, 25, -209.175]
  MoveL 1506 to (59.03, -111.65, -82.81) mm, rotated rx 56.95 ry 0 rz -151.03 deg; joints [119.96, -17.981, 55.621, -136.655, 46.682, 245.129, 25, -208.973]
  MoveL 1507 to (59.46, -112.26, -81.67) mm, rotated rx 56.95 ry 0 rz -151.03 deg; joints [119.951, -18.028, 55.599, -136.62, 46.626, 245.07, 25, -208.973]
  MoveL 1508 to (60.36, -112.5, -80.66) mm, rotated rx 57.04 ry 0 rz -150.99 deg; joints [119.926, -18.08, 55.548, -136.581, 46.539, 244.896, 25, -209.013]
  MoveL 1509 to (61.18, -112.49, -80.06) mm, rotated rx 57.31 ry 0 rz -150.67 deg; joints [119.91, -18.205, 55.5, -136.488, 46.404, 244.474, 25, -209.334]
  MoveL 1510 to (61.19, -112.52, -80) mm, rotated rx 58.25 ry 0 rz -150.38 deg; joints [119.881, -18.575, 55.389, -136.203, 46.04, 243.106, 25, -209.62]
  MoveL 1511 to (61.24, -113.39, -78.74) mm, rotated rx 58.81 ry 0 rz -150.55 deg; joints [119.85, -18.827, 55.283, -135.997, 45.765, 242.22, 25, -209.447]
  MoveL 1512 to (61.37, -113.79, -78.05) mm, rotated rx 58.81 ry 0 rz -150.55 deg; joints [119.848, -18.86, 55.273, -135.971, 45.733, 242.181, 25, -209.447]
  MoveL 1513 to (62, -114.24, -76.9) mm, rotated rx 58.93 ry 0 rz -150.54 deg; joints [119.832, -18.934, 55.223, -135.906, 45.635, 241.953, 25, -209.457]
  MoveL 1514 to (64.03, -114.71, -74.5) mm, rotated rx 59.98 ry 0 rz -149.88 deg; joints [119.785, -19.387, 55.013, -135.503, 45.133, 240.289, 25, -210.125]
  MoveL 1515 to (64.8, -115.27, -72.94) mm, rotated rx 60.89 ry 0 rz -149.61 deg; joints [119.758, -19.755, 54.841, -135.153, 44.734, 238.869, 25, -210.394]
  MoveL 1516 to (65.55, -115.43, -72.01) mm, rotated rx 60.89 ry 0 rz -149.61 deg; joints [119.743, -19.762, 54.803, -135.139, 44.693, 238.836, 25, -210.394]
  MoveL 1517 to (66.58, -115.27, -71.33) mm, rotated rx 60.95 ry 0 rz -149.54 deg; joints [119.721, -19.768, 54.749, -135.122, 44.639, 238.728, 25, -210.463]
  MoveL 1518 to (69.19, -114.39, -70.25) mm, rotated rx 61.42 ry 0 rz -148.39 deg; joints [119.707, -19.954, 54.648, -134.931, 44.427, 237.985, 25, -211.613]
  MoveL 1519 to (69.84, -114.17, -69.96) mm, rotated rx 61.55 ry 0 rz -148.08 deg; joints [119.705, -20.008, 54.621, -134.876, 44.369, 237.777, 25, -211.919]
  MoveL 1520 to (75.72, -112.02, -67.28) mm, rotated rx 62.7 ry 0 rz -145.47 deg; joints [119.68, -20.455, 54.361, -134.385, 43.857, 235.924, 25, -214.527]
  Set speed (16.7 mm/s)
  MoveL 1521 to (85.79, -126.66, -76.45) mm, rotated rx 62.7 ry 0 rz -145.47 deg; joints [118.912, -21.01, 54.772, -135.178, 43.303, 236.429, 25, -214.527]
  Set speed (1000.0 mm/s)
  MoveL 1522 to (70.78, -152.61, -30.8) mm, rotated rx 80.27 ry 0 rz -155.66 deg; joints [119.802, -25.234, 49.209, -125.355, 37.545, 206.551, 25, -204.341]
  Set speed (5.0 mm/s)
  MoveL 1523 to (62.66, -134.65, -27.42) mm, rotated rx 80.27 ry 0 rz -155.66 deg; joints [120.529, -24.583, 48.984, -125.013, 38.332, 206.495, 25, -204.341]
  Set speed (16.7 mm/s)
  MoveL 1524 to (60.97, -135.12, -28.83) mm, rotated rx 79.73 ry 0 rz -156.33 deg; joints [120.464, -24.516, 49.185, -125.358, 38.438, 207.448, 25, -203.671]
  MoveL 1525 to (60.92, -135.13, -28.89) mm, rotated rx 79.14 ry 0 rz -156.68 deg; joints [120.392, -24.412, 49.327, -125.689, 38.527, 208.418, 25, -203.318]
  MoveL 1526 to (60.25, -134.81, -31.58) mm, rotated rx 78.09 ry 0 rz -156.88 deg; joints [120.278, -24.264, 49.702, -126.342, 38.752, 210.237, 25, -203.125]
  Set speed (16.7 mm/s)
  MoveL 1527 to (67.93, -152.81, -35.71) mm, rotated rx 78.09 ry 0 rz -156.88 deg; joints [119.541, -24.912, 49.954, -126.755, 37.98, 210.364, 25, -203.125]
  Set speed (1000.0 mm/s)
  MoveL 1528 to (62.13, -154.29, -39.73) mm, rotated rx 77.4 ry 0 rz -158.11 deg; joints [119.5, -24.897, 50.341, -127.211, 38.193, 211.611, 25, -201.888]
  Set speed (5.0 mm/s)
  MoveL 1529 to (54.86, -136.18, -35.37) mm, rotated rx 77.4 ry 0 rz -158.11 deg; joints [120.241, -24.249, 50.081, -126.776, 38.96, 211.464, 25, -201.888]
  Set speed (16.7 mm/s)
  MoveL 1530 to (54.31, -136.4, -35.4) mm, rotated rx 77.39 ry 0 rz -158.34 deg; joints [120.24, -24.247, 50.086, -126.783, 38.963, 211.486, 25, -201.66]
  MoveL 1531 to (53.04, -136.99, -35.06) mm, rotated rx 77.39 ry 0 rz -158.34 deg; joints [120.274, -24.322, 50.122, -126.708, 38.964, 211.408, 25, -201.66]
  MoveL 1532 to (52.22, -137.43, -34.53) mm, rotated rx 77.6 ry 0 rz -158.7 deg; joints [120.294, -24.354, 50.049, -126.58, 38.916, 211.047, 25, -201.298]
  MoveL 1533 to (45.37, -141.15, -28.72) mm, rotated rx 79.79 ry 0 rz -161.59 deg; joints [120.54, -24.678, 49.264, -125.192, 38.446, 207.213, 25, -198.409]
  MoveL 1534 to (45.01, -141.33, -28.39) mm, rotated rx 79.89 ry 0 rz -161.71 deg; joints [120.554, -24.695, 49.229, -125.123, 38.427, 207.034, 25, -198.292]
  MoveL 1535 to (42.69, -142.49, -26.11) mm, rotated rx 80.75 ry 0 rz -162.68 deg; joints [120.66, -24.799, 48.911, -124.571, 38.265, 205.525, 25, -197.325]
  MoveL 1536 to (42.3, -142.7, -25.61) mm, rotated rx 80.75 ry 0 rz -162.68 deg; joints [120.675, -24.825, 48.909, -124.526, 38.26, 205.476, 25, -197.325]
  MoveL 1537 to (42.08, -142.83, -25.21) mm, rotated rx 80.9 ry 0 rz -162.77 deg; joints [120.694, -24.842, 48.852, -124.428, 38.233, 205.207, 25, -197.226]
  MoveL 1538 to (40.3, -143.93, -21.61) mm, rotated rx 82.23 ry 0 rz -163.52 deg; joints [120.872, -24.979, 48.347, -123.564, 38.009, 202.869, 25, -196.478]
  MoveL 1539 to (37.44, -145.06, -19.09) mm, rotated rx 83.46 ry 0 rz -164.91 deg; joints [121.023, -25.047, 47.878, -122.829, 37.831, 200.784, 25, -195.091]
  MoveL 1540 to (37.01, -145.23, -18.58) mm, rotated rx 83.46 ry 0 rz -164.91 deg; joints [121.039, -25.072, 47.876, -122.783, 37.829, 200.734, 25, -195.091]
  MoveL 1541 to (36.66, -145.4, -17.96) mm, rotated rx 83.58 ry 0 rz -164.99 deg; joints [121.064, -25.091, 47.827, -122.684, 37.812, 200.505, 25, -195.013]
  MoveL 1542 to (35.62, -145.92, -15.58) mm, rotated rx 84.48 ry 0 rz -165.42 deg; joints [121.199, -25.149, 47.471, -122.095, 37.695, 198.918, 25, -194.579]
  MoveL 1543 to (33.5, -146.58, -14.11) mm, rotated rx 85.43 ry 0 rz -166.6 deg; joints [121.313, -25.153, 47.1, -121.567, 37.588, 197.356, 25, -193.397]
  MoveL 1544 to (33.07, -146.71, -13.74) mm, rotated rx 85.49 ry 0 rz -166.67 deg; joints [121.332, -25.17, 47.08, -121.507, 37.583, 197.234, 25, -193.335]
  MoveL 1545 to (31.61, -147.19, -11.93) mm, rotated rx 86.07 ry 0 rz -167.14 deg; joints [121.435, -25.209, 46.846, -121.101, 37.523, 196.187, 25, -192.857]
  MoveL 1546 to (31.23, -147.3, -11.66) mm, rotated rx 86.3 ry 0 rz -167.42 deg; joints [121.461, -25.2, 46.754, -120.982, 37.501, 195.819, 25, -192.58]
  MoveL 1547 to (25.25, -148.78, -5.86) mm, rotated rx 88.47 ry 0 rz -169.71 deg; joints [121.836, -25.253, 45.872, -119.561, 37.332, 192.035, 25, -190.286]
  MoveL 1548 to (24.36, -148.99, -4.06) mm, rotated rx 88.49 ry 0 rz -169.68 deg; joints [121.888, -25.301, 45.836, -119.415, 37.333, 191.853, 25, -190.317]
  MoveL 1549 to (24.52, -148.98, -3.15) mm, rotated rx 88.5 ry 0 rz -169.67 deg; joints [121.9, -25.295, 45.798, -119.367, 37.327, 191.788, 25, -190.331]
  MoveL 1550 to (25.82, -148.79, -1.69) mm, rotated rx 88.52 ry 0 rz -169.64 deg; joints [121.896, -25.238, 45.705, -119.33, 37.306, 191.719, 25, -190.361]
  MoveL 1551 to (27.78, -148.44, -1.42) mm, rotated rx 88.54 ry 0 rz -169.61 deg; joints [121.86, -25.147, 45.63, -119.383, 37.284, 191.749, 25, -190.391]
  MoveL 1552 to (31.01, -147.79, -2.17) mm, rotated rx 88.25 ry 0 rz -168.36 deg; joints [121.808, -25.146, 45.749, -119.569, 37.301, 192.246, 25, -191.638]
  MoveL 1553 to (33.69, -147.2, -2.25) mm, rotated rx 88.2 ry 0 rz -167.14 deg; joints [121.81, -25.168, 45.783, -119.581, 37.308, 192.314, 25, -192.857]
  MoveL 1554 to (34.44, -147.02, -2.4) mm, rotated rx 88.2 ry 0 rz -167.14 deg; joints [121.79, -25.131, 45.764, -119.62, 37.301, 192.355, 25, -192.857]
  MoveL 1555 to (34.9, -146.91, -2.57) mm, rotated rx 88.13 ry 0 rz -166.96 deg; joints [121.779, -25.13, 45.791, -119.663, 37.305, 192.469, 25, -193.036]
  MoveL 1556 to (35.62, -146.73, -3) mm, rotated rx 88.13 ry 0 rz -166.96 deg; joints [121.756, -25.095, 45.782, -119.715, 37.3, 192.525, 25, -193.036]
  MoveL 1557 to (39.46, -145.64, -6.33) mm, rotated rx 86.87 ry 0 rz -165.45 deg; joints [121.535, -25.073, 46.299, -120.54, 37.392, 194.728, 25, -194.549]
  MoveL 1558 to (41.08, -145.14, -7.17) mm, rotated rx 86.44 ry 0 rz -164.63 deg; joints [121.478, -25.084, 46.478, -120.787, 37.432, 195.443, 25, -195.366]
  Set speed (16.7 mm/s)
  MoveL 1559 to (46.37, -164.39, -8.41) mm, rotated rx 86.44 ry 0 rz -164.63 deg; joints [120.79, -25.727, 46.626, -120.906, 36.627, 195.282, 25, -195.366]
  Set speed (1000.0 mm/s)
  MoveL 1560 to (62.65, -157.67, -21.45) mm, rotated rx 82.12 ry 0 rz -158.83 deg; joints [120.095, -25.462, 48.376, -123.893, 37.162, 203.012, 25, -201.171]
  Set speed (5.0 mm/s)
  MoveL 1561 to (55.49, -139.2, -18.7) mm, rotated rx 82.12 ry 0 rz -158.83 deg; joints [120.811, -24.813, 48.174, -123.62, 37.958, 203.022, 25, -201.171]
  Set speed (16.7 mm/s)
  MoveL 1562 to (56.32, -138.78, -19.37) mm, rotated rx 81.86 ry 0 rz -158.48 deg; joints [120.776, -24.79, 48.271, -123.784, 37.998, 203.467, 25, -201.523]
  MoveL 1563 to (56.8, -138.51, -19.87) mm, rotated rx 81.77 ry 0 rz -158.38 deg; joints [120.754, -24.764, 48.304, -123.87, 38.014, 203.658, 25, -201.616]
  MoveL 1564 to (57.53, -138.1, -20.62) mm, rotated rx 81.45 ry 0 rz -158.03 deg; joints [120.714, -24.739, 48.426, -124.068, 38.067, 204.21, 25, -201.974]
  MoveL 1565 to (57.56, -138.08, -20.68) mm, rotated rx 81.26 ry 0 rz -156.98 deg; joints [120.754, -24.856, 48.57, -124.054, 38.112, 204.401, 25, -203.017]
  MoveL 1566 to (58.55, -137.73, -20.22) mm, rotated rx 81.44 ry 0 rz -156.58 deg; joints [120.777, -24.874, 48.504, -123.941, 38.082, 204.093, 25, -203.419]
  MoveL 1567 to (60.3, -136.98, -20.17) mm, rotated rx 81.44 ry 0 rz -156.58 deg; joints [120.735, -24.781, 48.441, -124.017, 38.068, 204.169, 25, -203.419]
  MoveL 1568 to (61.39, -136.38, -20.98) mm, rotated rx 81.41 ry 0 rz -156.5 deg; joints [120.701, -24.721, 48.442, -124.118, 38.075, 204.308, 25, -203.497]
  MoveL 1569 to (63.29, -135.06, -23.68) mm, rotated rx 80.37 ry 0 rz -155.63 deg; joints [120.569, -24.611, 48.83, -124.781, 38.258, 206.119, 25, -204.368]
  Set speed (16.7 mm/s)
  MoveL 1570 to (71.42, -153.02, -27.03) mm, rotated rx 80.37 ry 0 rz -155.63 deg; joints [119.843, -25.261, 49.054, -125.115, 37.47, 206.169, 25, -204.368]
  Set speed (1000.0 mm/s)
  MoveL 1571 to (90.43, -139.29, -40.79) mm, rotated rx 75.42 ry 0 rz -147.31 deg; joints [119.33, -24.579, 50.891, -128.27, 38.603, 214.853, 25, -212.692]
  Set speed (5.0 mm/s)
  MoveL 1572 to (79.98, -123, -35.75) mm, rotated rx 75.42 ry 0 rz -147.31 deg; joints [120.079, -23.936, 50.608, -127.776, 39.352, 214.648, 25, -212.692]
  Set speed (16.7 mm/s)
  MoveL 1573 to (83.77, -119.93, -37.51) mm, rotated rx 74.73 ry 0 rz -145.41 deg; joints [120.021, -23.807, 50.84, -128.188, 39.534, 215.836, 25, -214.592]
  Set speed (16.7 mm/s)
  MoveL 1574 to (94.73, -135.81, -42.78) mm, rotated rx 74.73 ry 0 rz -145.41 deg; joints [119.27, -24.447, 51.131, -128.702, 38.792, 216.061, 25, -214.592]
  Set speed (1000.0 mm/s)
  MoveL 1575 to (92.71, -135.53, -47.8) mm, rotated rx 74.61 ry 0 rz -145.59 deg; joints [119.249, -24.395, 51.337, -128.975, 38.94, 216.524, 25, -214.405]
  Set speed (5.0 mm/s)
  MoveL 1576 to (81.81, -119.62, -42.49) mm, rotated rx 74.61 ry 0 rz -145.59 deg; joints [120.001, -23.753, 51.044, -128.454, 39.68, 216.292, 25, -214.405]
  Set speed (16.7 mm/s)
  MoveL 1577 to (77.51, -122.51, -42.31) mm, rotated rx 74.68 ry 0 rz -147.64 deg; joints [120.007, -23.768, 51.02, -128.411, 39.66, 216.168, 25, -212.356]
  MoveL 1578 to (76.94, -122.89, -42.25) mm, rotated rx 74.7 ry 0 rz -147.85 deg; joints [120.012, -23.78, 51.019, -128.393, 39.655, 216.127, 25, -212.149]
  MoveL 1579 to (72.84, -125.43, -42.04) mm, rotated rx 74.78 ry 0 rz -149.81 deg; joints [120.015, -23.79, 50.986, -128.348, 39.631, 215.985, 25, -210.19]
  MoveL 1580 to (72.06, -125.92, -41.94) mm, rotated rx 74.82 ry 0 rz -150.09 deg; joints [120.023, -23.808, 50.981, -128.318, 39.622, 215.916, 25, -209.909]
  MoveL 1581 to (66.64, -129.33, -40.5) mm, rotated rx 75.37 ry 0 rz -152.52 deg; joints [120.073, -23.928, 50.803, -127.978, 39.473, 214.954, 25, -207.484]
  MoveL 1582 to (63.46, -130.9, -40.56) mm, rotated rx 75.37 ry 0 rz -154.14 deg; joints [120.059, -23.898, 50.786, -128.006, 39.472, 214.983, 25, -205.857]
  MoveL 1583 to (62.54, -131.38, -40.43) mm, rotated rx 75.41 ry 0 rz -154.37 deg; joints [120.073, -23.929, 50.786, -127.961, 39.463, 214.894, 25, -205.628]
  MoveL 1584 to (62.02, -131.68, -40.24) mm, rotated rx 75.41 ry 0 rz -154.37 deg; joints [120.087, -23.962, 50.801, -127.928, 39.461, 214.859, 25, -205.628]
  MoveL 1585 to (56.11, -135.18, -37.23) mm, rotated rx 76.59 ry 0 rz -157.05 deg; joints [120.191, -24.175, 50.396, -127.214, 39.158, 212.812, 25, -202.946]
  Set speed (16.7 mm/s)
  MoveL 1586 to (63.69, -153.09, -41.87) mm, rotated rx 76.59 ry 0 rz -157.05 deg; joints [119.446, -24.823, 50.666, -127.674, 38.397, 212.982, 25, -202.946]
  Set speed (1000.0 mm/s)
  MoveL 1587 to (68.16, -152.61, -36.11) mm, rotated rx 76.99 ry 0 rz -155.76 deg; joints [119.512, -24.926, 50.372, -127.2, 38.203, 212.018, 25, -204.241]
  Set speed (5.0 mm/s)
  MoveL 1588 to (60.16, -134.85, -31.61) mm, rotated rx 76.99 ry 0 rz -155.76 deg; joints [120.255, -24.278, 50.108, -126.758, 38.968, 211.863, 25, -204.241]
  Set speed (16.7 mm/s)
  MoveL 1589 to (61.76, -134.22, -31.26) mm, rotated rx 77.13 ry 0 rz -155.09 deg; joints [120.268, -24.301, 50.06, -126.674, 38.935, 211.626, 25, -204.909]
  MoveL 1590 to (62.6, -133.84, -31.24) mm, rotated rx 77.13 ry 0 rz -155.09 deg; joints [120.247, -24.255, 50.029, -126.711, 38.93, 211.663, 25, -204.909]
  MoveL 1591 to (63.41, -133.42, -31.39) mm, rotated rx 77.07 ry 0 rz -154.74 deg; joints [120.242, -24.246, 50.049, -126.747, 38.943, 211.762, 25, -205.263]
  MoveL 1592 to (70.32, -129.46, -33.2) mm, rotated rx 76.39 ry 0 rz -151.23 deg; joints [120.2, -24.187, 50.324, -127.121, 39.113, 212.9, 25, -208.773]
  MoveL 1593 to (72.05, -128.64, -32.68) mm, rotated rx 76.59 ry 0 rz -150.48 deg; joints [120.219, -24.222, 50.253, -126.998, 39.064, 212.549, 25, -209.515]
  MoveL 1594 to (72.71, -128.29, -32.59) mm, rotated rx 76.59 ry 0 rz -150.48 deg; joints [120.203, -24.185, 50.226, -127.024, 39.058, 212.574, 25, -209.515]
  MoveL 1595 to (73.24, -127.99, -32.6) mm, rotated rx 76.58 ry 0 rz -150.25 deg; joints [120.202, -24.184, 50.229, -127.028, 39.06, 212.586, 25, -209.752]
  MoveL 1596 to (78.41, -124.63, -33.57) mm, rotated rx 76.22 ry 0 rz -147.98 deg; joints [120.161, -24.105, 50.345, -127.266, 39.147, 213.232, 25, -212.018]
  Set speed (16.7 mm/s)
  MoveL 1597 to (88.71, -141.1, -38.33) mm, rotated rx 76.22 ry 0 rz -147.98 deg; joints [119.415, -24.75, 50.618, -127.733, 38.39, 213.412, 25, -212.018]
  Set speed (1000.0 mm/s)
  MoveL 1598 to (102.21, -137.05, -2.99) mm, rotated rx 89.52 ry 0 rz -143.94 deg; joints [121.284, -25.714, 45.423, -119.031, 36.434, 190.085, 25, -216.056]
  Set speed (5.0 mm/s)
  MoveL 1599 to (90.44, -120.88, -2.82) mm, rotated rx 89.52 ry 0 rz -143.94 deg; joints [121.949, -25.079, 45.315, -119.014, 37.236, 190.347, 25, -216.056]
  Set speed (16.7 mm/s)
  MoveL 1600 to (88.38, -122.31, -6) mm, rotated rx 88.31 ry 0 rz -144.89 deg; joints [121.73, -25.077, 45.813, -119.797, 37.303, 192.438, 25, -215.106]
  MoveL 1601 to (87.92, -122.62, -6.51) mm, rotated rx 88.31 ry 0 rz -144.89 deg; joints [121.735, -25.103, 45.847, -119.801, 37.311, 192.446, 25, -215.106]
  MoveL 1602 to (87.39, -122.97, -6.95) mm, rotated rx 88.15 ry 0 rz -145.14 deg; joints [121.705, -25.1, 45.915, -119.909, 37.322, 192.735, 25, -214.862]
  MoveL 1603 to (86.92, -123.29, -7.24) mm, rotated rx 88.15 ry 0 rz -145.14 deg; joints [121.714, -25.127, 45.943, -119.902, 37.33, 192.729, 25, -214.862]
  MoveL 1604 to (84.87, -124.65, -8.12) mm, rotated rx 87.81 ry 0 rz -146.07 deg; joints [121.655, -25.122, 46.079, -120.119, 37.353, 193.31, 25, -213.93]
  MoveL 1605 to (83.39, -125.52, -9.9) mm, rotated rx 86.9 ry 0 rz -147.08 deg; joints [121.487, -25.057, 46.401, -120.721, 37.413, 194.902, 25, -212.916]
  MoveL 1606 to (82.93, -125.79, -10.4) mm, rotated rx 86.82 ry 0 rz -147.17 deg; joints [121.476, -25.069, 46.454, -120.777, 37.425, 195.053, 25, -212.832]
  MoveL 1607 to (80.75, -127.03, -12.24) mm, rotated rx 86.11 ry 0 rz -148.12 deg; joints [121.36, -25.045, 46.736, -121.235, 37.491, 196.277, 25, -211.879]
  MoveL 1608 to (80.17, -127.37, -12.59) mm, rotated rx 86.11 ry 0 rz -148.12 deg; joints [121.37, -25.076, 46.768, -121.226, 37.5, 196.27, 25, -211.879]
  MoveL 1609 to (79.49, -127.77, -12.82) mm, rotated rx 86.07 ry 0 rz -148.25 deg; joints [121.372, -25.096, 46.804, -121.242, 37.509, 196.336, 25, -211.75]
  MoveL 1610 to (77.53, -128.92, -13.15) mm, rotated rx 85.95 ry 0 rz -149.12 deg; joints [121.352, -25.091, 46.854, -121.324, 37.522, 196.555, 25, -210.885]
  MoveL 1611 to (77.4, -129, -13.17) mm, rotated rx 85.63 ry 0 rz -149.74 deg; joints [121.278, -25.007, 46.907, -121.55, 37.535, 197.122, 25, -210.256]
  MoveL 1612 to (75.72, -129.77, -15.23) mm, rotated rx 84.84 ry 0 rz -150.45 deg; joints [121.155, -24.968, 47.218, -122.061, 37.622, 198.493, 25, -209.552]
  MoveL 1613 to (74.71, -130.28, -15.95) mm, rotated rx 84.84 ry 0 rz -150.45 deg; joints [121.171, -25.019, 47.277, -122.052, 37.639, 198.49, 25, -209.552]
  MoveL 1614 to (74.3, -130.49, -16.09) mm, rotated rx 84.79 ry 0 rz -150.62 deg; joints [121.163, -25.017, 47.298, -122.087, 37.645, 198.582, 25, -209.378]
  MoveL 1615 to (73.34, -131.02, -16.17) mm, rotated rx 84.79 ry 0 rz -150.62 deg; joints [121.186, -25.069, 47.335, -122.046, 37.655, 198.541, 25, -209.378]
  MoveL 1616 to (72.39, -131.56, -16.01) mm, rotated rx 84.85 ry 0 rz -151.04 deg; joints [121.196, -25.072, 47.311, -122.006, 37.648, 198.435, 25, -208.962]
  MoveL 1617 to (72.28, -131.59, -16.02) mm, rotated rx 84.17 ry 0 rz -152.14 deg; joints [121.054, -24.906, 47.434, -122.468, 37.692, 199.629, 25, -207.864]
  MoveL 1618 to (71.42, -131.71, -18.79) mm, rotated rx 83.11 ry 0 rz -152.45 deg; joints [120.899, -24.831, 47.846, -123.156, 37.835, 201.482, 25, -207.553]
  MoveL 1619 to (71.39, -131.76, -18.67) mm, rotated rx 82.23 ry 0 rz -152.23 deg; joints [120.816, -24.805, 48.129, -123.574, 37.942, 202.854, 25, -207.77]
  MoveL 1620 to (72.97, -130.61, -20.61) mm, rotated rx 81.49 ry 0 rz -151.49 deg; joints [120.716, -24.737, 48.411, -124.051, 38.061, 204.15, 25, -208.509]
  MoveL 1621 to (73.3, -130.32, -21.19) mm, rotated rx 81.49 ry 0 rz -151.49 deg; joints [120.701, -24.711, 48.415, -124.1, 38.065, 204.204, 25, -208.509]
  MoveL 1622 to (73.51, -130.11, -21.78) mm, rotated rx 81.38 ry 0 rz -151.43 deg; joints [120.68, -24.692, 48.46, -124.19, 38.086, 204.413, 25, -208.565]
  MoveL 1623 to (73.91, -129.59, -23.41) mm, rotated rx 80.76 ry 0 rz -151.21 deg; joints [120.6, -24.626, 48.695, -124.59, 38.196, 205.505, 25, -208.795]
  MoveL 1624 to (73.94, -129.56, -23.52) mm, rotated rx 80.1 ry 0 rz -150.41 deg; joints [120.58, -24.668, 48.956, -124.841, 38.306, 206.474, 25, -209.593]
  MoveL 1625 to (75.23, -128.78, -23.7) mm, rotated rx 80.03 ry 0 rz -149.83 deg; joints [120.571, -24.66, 48.983, -124.887, 38.319, 206.599, 25, -210.173]
  MoveL 1626 to (75.71, -128.49, -23.8) mm, rotated rx 80 ry 0 rz -149.68 deg; joints [120.564, -24.648, 48.989, -124.914, 38.324, 206.658, 25, -210.325]
  MoveL 1627 to (77.54, -127.24, -24.56) mm, rotated rx 79.75 ry 0 rz -148.97 deg; joints [120.524, -24.598, 49.073, -125.095, 38.371, 207.121, 25, -211.031]
  MoveL 1628 to (79.37, -126.18, -24.21) mm, rotated rx 79.84 ry 0 rz -147.68 deg; joints [120.563, -24.671, 49.076, -124.981, 38.36, 206.906, 25, -212.315]
  MoveL 1629 to (79.85, -125.89, -24.17) mm, rotated rx 79.84 ry 0 rz -147.58 deg; joints [120.558, -24.658, 49.065, -124.988, 38.357, 206.908, 25, -212.425]
  MoveL 1630 to (80.62, -125.37, -24.31) mm, rotated rx 79.84 ry 0 rz -147.58 deg; joints [120.536, -24.611, 49.039, -125.034, 38.353, 206.955, 25, -212.425]
  MoveL 1631 to (84.37, -122.54, -25.92) mm, rotated rx 79.22 ry 0 rz -145.77 deg; joints [120.463, -24.533, 49.268, -125.428, 38.475, 208.042, 25, -214.229]
  MoveL 1632 to (85.93, -121.52, -25.55) mm, rotated rx 79.33 ry 0 rz -144.55 deg; joints [120.505, -24.613, 49.268, -125.301, 38.461, 207.796, 25, -215.448]
  MoveL 1633 to (85.95, -121.5, -25.53) mm, rotated rx 79.99 ry 0 rz -143.81 deg; joints [120.609, -24.771, 49.137, -124.89, 38.372, 206.664, 25, -216.194]
  MoveL 1634 to (87.01, -121.36, -22.54) mm, rotated rx 81.14 ry 0 rz -143.45 deg; joints [120.752, -24.899, 48.709, -124.158, 38.164, 204.658, 25, -216.554]
  MoveL 1635 to (87.23, -121.31, -21.95) mm, rotated rx 81.33 ry 0 rz -143.38 deg; joints [120.777, -24.918, 48.632, -124.03, 38.13, 204.314, 25, -216.623]
  MoveL 1636 to (87.97, -120.98, -20.84) mm, rotated rx 81.33 ry 0 rz -143.38 deg; joints [120.772, -24.888, 48.572, -124.005, 38.109, 204.279, 25, -216.623]
  MoveL 1637 to (90.1, -119.71, -18.88) mm, rotated rx 82.08 ry 0 rz -142.44 deg; joints [120.872, -24.957, 48.288, -123.523, 37.988, 202.97, 25, -217.564]
  MoveL 1638 to (90.09, -119.72, -18.86) mm, rotated rx 82.81 ry 0 rz -142.08 deg; joints [120.973, -25.051, 48.097, -123.113, 37.909, 201.77, 25, -217.918]
  MoveL 1639 to (90.21, -119.83, -17.57) mm, rotated rx 83.3 ry 0 rz -142.07 deg; joints [121.043, -25.089, 47.906, -122.793, 37.839, 200.907, 25, -217.928]
  MoveL 1640 to (90.47, -119.79, -16.57) mm, rotated rx 83.3 ry 0 rz -142.07 deg; joints [121.049, -25.084, 47.867, -122.75, 37.826, 200.856, 25, -217.928]
  MoveL 1641 to (91.5, -119.19, -15.17) mm, rotated rx 83.41 ry 0 rz -142.02 deg; joints [121.054, -25.047, 47.757, -122.666, 37.79, 200.645, 25, -217.977]
  MoveL 1642 to (92.23, -118.67, -14.67) mm, rotated rx 83.6 ry 0 rz -141.68 deg; joints [121.082, -25.06, 47.683, -122.543, 37.766, 200.315, 25, -218.317]
  MoveL 1643 to (92.16, -118.73, -14.72) mm, rotated rx 84.96 ry 0 rz -141.41 deg; joints [121.263, -25.163, 47.287, -121.812, 37.64, 198.109, 25, -218.589]
  MoveL 1644 to (91.86, -119.04, -14.06) mm, rotated rx 85.06 ry 0 rz -141.48 deg; joints [121.288, -25.181, 47.244, -121.719, 37.628, 197.91, 25, -218.521]
  MoveL 1645 to (91.17, -119.81, -11.87) mm, rotated rx 85.89 ry 0 rz -141.87 deg; joints [121.421, -25.219, 46.91, -121.174, 37.539, 196.449, 25, -218.13]
  MoveL 1646 to (91.03, -119.98, -11.18) mm, rotated rx 85.96 ry 0 rz -141.89 deg; joints [121.443, -25.232, 46.871, -121.095, 37.53, 196.289, 25, -218.114]
  MoveL 1647 to (91.3, -119.93, -9.43) mm, rotated rx 85.96 ry 0 rz -141.89 deg; joints [121.46, -25.225, 46.807, -121.013, 37.514, 196.194, 25, -218.114]
  MoveL 1648 to (93.2, -118.68, -5.31) mm, rotated rx 87.53 ry 0 rz -141.03 deg; joints [121.725, -25.266, 46.172, -119.994, 37.384, 193.468, 25, -218.973]
  MoveL 1649 to (93.25, -118.66, -5.43) mm, rotated rx 88.75 ry 0 rz -141.35 deg; joints [121.874, -25.233, 45.751, -119.409, 37.312, 191.572, 25, -218.651]
  MoveL 1650 to (92.38, -119.37, -4.75) mm, rotated rx 89.01 ry 0 rz -141.78 deg; joints [121.92, -25.234, 45.645, -119.243, 37.297, 191.128, 25, -218.224]
  MoveL 1651 to (91.89, -119.77, -4.26) mm, rotated rx 89.1 ry 0 rz -141.89 deg; joints [121.948, -25.251, 45.608, -119.154, 37.295, 190.935, 25, -218.114]
  MoveL 1652 to (90.37, -120.94, -2.83) mm, rotated rx 89.69 ry 0 rz -142.66 deg; joints [122.052, -25.242, 45.365, -118.788, 37.267, 189.937, 25, -217.336]
  Set speed (16.7 mm/s)
  MoveL 1653 to (102.5, -136.84, -2.93) mm, rotated rx 89.69 ry 0 rz -142.66 deg; joints [121.388, -25.878, 45.471, -118.795, 36.464, 189.664, 25, -217.336]
  Set speed (1000.0 mm/s)
  MoveL 1654 to (69.67, -151.25, 38.86) mm, rotated rx 103.85 ry 0 rz -154.81 deg; joints [124.723, -24.538, 39.046, -109.874, 37.278, 165.584, 25, -205.188]
  Set speed (5.0 mm/s)
  MoveL 1655 to (61.4, -133.67, 34.08) mm, rotated rx 103.85 ry 0 rz -154.81 deg; joints [125.251, -23.983, 39.127, -110.286, 37.976, 166.275, 25, -205.188]
  Set speed (16.7 mm/s)
  MoveL 1656 to (60.3, -134, 34.77) mm, rotated rx 104.12 ry 0 rz -155.26 deg; joints [125.321, -23.94, 39.004, -110.142, 38.012, 165.847, 25, -204.745]
  MoveL 1657 to (60.33, -134.01, 34.7) mm, rotated rx 104.01 ry 0 rz -156.39 deg; joints [125.229, -23.829, 38.96, -110.286, 37.951, 166.102, 25, -203.612]
  MoveL 1658 to (56.93, -136.29, 31.42) mm, rotated rx 102.74 ry 0 rz -157.95 deg; joints [124.9, -24.029, 39.541, -110.975, 37.788, 168.137, 25, -202.048]
  MoveL 1659 to (56.94, -136.29, 31.37) mm, rotated rx 101.33 ry 0 rz -158.02 deg; joints [124.613, -24.183, 40.042, -111.6, 37.657, 170.241, 25, -201.982]
  MoveL 1660 to (60.3, -135.6, 27.99) mm, rotated rx 100.02 ry 0 rz -156.71 deg; joints [124.287, -24.359, 40.634, -112.344, 37.523, 172.376, 25, -203.286]
  MoveL 1661 to (61.36, -135.26, 27.32) mm, rotated rx 99.64 ry 0 rz -156.14 deg; joints [124.209, -24.42, 40.806, -112.536, 37.495, 172.973, 25, -203.857]
  MoveL 1662 to (62.08, -135.09, 26.55) mm, rotated rx 99.64 ry 0 rz -156.14 deg; joints [124.177, -24.395, 40.812, -112.599, 37.479, 173.041, 25, -203.857]
  MoveL 1663 to (69.88, -133.18, 13.65) mm, rotated rx 94.69 ry 0 rz -153.13 deg; joints [123.036, -24.87, 43.002, -115.573, 37.184, 181.297, 25, -206.873]
  MoveL 1664 to (70.2, -133.1, 12.83) mm, rotated rx 94.69 ry 0 rz -153.13 deg; joints [123.014, -24.86, 43.022, -115.627, 37.178, 181.357, 25, -206.873]
  MoveL 1665 to (69.89, -133.43, 10.9) mm, rotated rx 94.69 ry 0 rz -153.13 deg; joints [122.99, -24.89, 43.102, -115.708, 37.18, 181.449, 25, -206.873]
  MoveL 1666 to (69.52, -133.67, 10.31) mm, rotated rx 94.47 ry 0 rz -153.29 deg; joints [122.942, -24.905, 43.201, -115.849, 37.174, 181.833, 25, -206.709]
  MoveL 1667 to (68.72, -134.14, 9.53) mm, rotated rx 94.47 ry 0 rz -153.29 deg; joints [122.949, -24.951, 43.256, -115.853, 37.185, 181.841, 25, -206.709]
  MoveL 1668 to (62.93, -137.14, 6.34) mm, rotated rx 93.26 ry 0 rz -155.77 deg; joints [122.693, -25.019, 43.78, -116.615, 37.168, 183.905, 25, -204.232]
  MoveL 1669 to (62.6, -137.3, 6.11) mm, rotated rx 93.14 ry 0 rz -155.97 deg; joints [122.665, -25.017, 43.824, -116.694, 37.166, 184.116, 25, -204.025]
  MoveL 1670 to (57.66, -139.56, 2.56) mm, rotated rx 91.77 ry 0 rz -158.07 deg; joints [122.386, -25.067, 44.404, -117.567, 37.172, 186.464, 25, -201.93]
  Set speed (16.7 mm/s)
  MoveL 1671 to (65.13, -158.1, 3.18) mm, rotated rx 91.77 ry 0 rz -158.07 deg; joints [121.74, -25.694, 44.483, -117.506, 36.378, 186.125, 25, -201.93]
  Set speed (1000.0 mm/s)
  MoveL 1672 to (61.23, -159.61, 4.89) mm, rotated rx 91.82 ry 0 rz -158.19 deg; joints [121.862, -25.865, 44.522, -117.234, 36.419, 185.783, 25, -201.806]
  Set speed (5.0 mm/s)
  MoveL 1673 to (53.8, -141.05, 4.25) mm, rotated rx 91.82 ry 0 rz -158.19 deg; joints [122.509, -25.238, 44.444, -117.302, 37.215, 186.131, 25, -201.806]
  Set speed (16.7 mm/s)
  MoveL 1674 to (53.45, -141.12, 5.86) mm, rotated rx 92.43 ry 0 rz -158.33 deg; joints [122.632, -25.214, 44.183, -116.914, 37.211, 185.084, 25, -201.669]
  MoveL 1675 to (53.42, -141.12, 5.84) mm, rotated rx 93.06 ry 0 rz -158.84 deg; joints [122.705, -25.131, 43.93, -116.65, 37.195, 184.148, 25, -201.164]
  MoveL 1676 to (50.11, -142.26, 7.61) mm, rotated rx 93.74 ry 0 rz -160.17 deg; joints [122.845, -25.097, 43.64, -116.226, 37.2, 182.999, 25, -199.831]
  MoveL 1677 to (49.43, -142.47, 8.08) mm, rotated rx 93.84 ry 0 rz -160.31 deg; joints [122.877, -25.105, 43.599, -116.139, 37.206, 182.802, 25, -199.69]
  MoveL 1678 to (46.88, -143.14, 10.85) mm, rotated rx 94.76 ry 0 rz -161.17 deg; joints [123.09, -25.063, 43.197, -115.53, 37.231, 181.196, 25, -198.833]
  MoveL 1679 to (43.15, -144.21, 12.26) mm, rotated rx 95.55 ry 0 rz -163.01 deg; joints [123.228, -24.966, 42.847, -115.113, 37.242, 179.94, 25, -196.987]
  MoveL 1680 to (42.56, -144.35, 12.56) mm, rotated rx 95.61 ry 0 rz -163.12 deg; joints [123.251, -24.975, 42.826, -115.058, 37.249, 179.822, 25, -196.879]
  MoveL 1681 to (42.42, -144.38, 12.73) mm, rotated rx 95.12 ry 0 rz -164.53 deg; joints [123.089, -24.84, 42.879, -115.419, 37.189, 180.693, 25, -195.466]
  MoveL 1682 to (42.22, -144.5, 11.97) mm, rotated rx 94.8 ry 0 rz -164.63 deg; joints [123.018, -24.861, 43.018, -115.619, 37.179, 181.244, 25, -195.371]
  MoveL 1683 to (41.24, -145.04, 8.08) mm, rotated rx 93.32 ry 0 rz -165.04 deg; joints [122.704, -24.949, 43.657, -116.544, 37.154, 183.755, 25, -194.957]
  MoveL 1684 to (41.22, -145.05, 8.08) mm, rotated rx 92.4 ry 0 rz -164.81 deg; joints [122.568, -25.013, 43.99, -116.981, 37.16, 185.174, 25, -195.192]
  MoveL 1685 to (42.7, -144.71, 6.56) mm, rotated rx 91.82 ry 0 rz -164.23 deg; joints [122.45, -25.036, 44.236, -117.348, 37.163, 186.163, 25, -195.767]
  MoveL 1686 to (43.29, -144.57, 5.76) mm, rotated rx 91.64 ry 0 rz -164.1 deg; joints [122.402, -25.031, 44.317, -117.493, 37.162, 186.508, 25, -195.897]
  MoveL 1687 to (45.2, -144.07, 2.42) mm, rotated rx 90.03 ry 0 rz -162.91 deg; joints [122.129, -25.123, 45.001, -118.433, 37.213, 189.179, 25, -197.088]
  MoveL 1688 to (47.5, -143.35, 1.53) mm, rotated rx 89.69 ry 0 rz -162 deg; joints [122.064, -25.128, 45.144, -118.653, 37.225, 189.769, 25, -198.002]
  MoveL 1689 to (48.44, -143.04, 0.99) mm, rotated rx 89.56 ry 0 rz -161.77 deg; joints [122.027, -25.111, 45.195, -118.765, 37.227, 190.028, 25, -198.232]
  MoveL 1690 to (53.7, -141.11, -3.5) mm, rotated rx 87.93 ry 0 rz -159.76 deg; joints [121.721, -25.094, 45.865, -119.843, 37.313, 192.871, 25, -200.238]
  MoveL 1691 to (54.37, -140.82, -4.48) mm, rotated rx 87.93 ry 0 rz -159.76 deg; joints [121.691, -25.059, 45.875, -119.924, 37.311, 192.96, 25, -200.238]
  MoveL 1692 to (54.55, -140.74, -4.93) mm, rotated rx 87.76 ry 0 rz -159.69 deg; joints [121.661, -25.056, 45.945, -120.036, 37.323, 193.257, 25, -200.31]
  MoveL 1693 to (54.71, -140.65, -5.7) mm, rotated rx 87.76 ry 0 rz -159.69 deg; joints [121.646, -25.046, 45.964, -120.084, 37.326, 193.311, 25, -200.31]
  MoveL 1694 to (54.93, -140.34, -9.65) mm, rotated rx 86.26 ry 0 rz -159.57 deg; joints [121.391, -25.008, 46.574, -121.065, 37.451, 195.932, 25, -200.43]
  MoveL 1695 to (56.36, -139.38, -14.28) mm, rotated rx 84.26 ry 0 rz -158.88 deg; joints [121.085, -24.922, 47.354, -122.332, 37.665, 199.387, 25, -201.119]
  Set speed (16.7 mm/s)
  MoveL 1696 to (63.53, -157.94, -16.28) mm, rotated rx 84.26 ry 0 rz -158.88 deg; joints [120.383, -25.569, 47.529, -122.532, 36.863, 199.306, 25, -201.119]
  Set speed (1000.0 mm/s)
  MoveL 1697 to (46.92, -164.25, -8.17) mm, rotated rx 87.45 ry 0 rz -163.24 deg; joints [121.011, -25.918, 46.403, -120.208, 36.595, 193.495, 25, -196.76]
  Set speed (5.0 mm/s)
  MoveL 1698 to (41.16, -145.12, -7.28) mm, rotated rx 87.45 ry 0 rz -163.24 deg; joints [121.692, -25.274, 46.269, -120.125, 37.402, 193.693, 25, -196.76]
  Set speed (16.7 mm/s)
  MoveL 1699 to (40.47, -145.44, -4.09) mm, rotated rx 88.66 ry 0 rz -163.52 deg; joints [121.906, -25.288, 45.771, -119.338, 37.322, 191.588, 25, -196.475]
  MoveL 1700 to (37.19, -146.37, -0.4) mm, rotated rx 90.49 ry 0 rz -165.05 deg; joints [122.216, -25.248, 45.028, -118.239, 37.238, 188.514, 25, -194.955]
  MoveL 1701 to (37.63, -146.26, -0.79) mm, rotated rx 90.49 ry 0 rz -165.05 deg; joints [122.2, -25.227, 45.028, -118.277, 37.234, 188.555, 25, -194.955]
  MoveL 1702 to (37.24, -146.36, -0.52) mm, rotated rx 90.59 ry 0 rz -165.2 deg; joints [122.219, -25.225, 44.985, -118.212, 37.231, 188.38, 25, -194.802]
  MoveL 1703 to (33.99, -147.13, 2.15) mm, rotated rx 91.55 ry 0 rz -166.4 deg; joints [122.413, -25.21, 44.578, -117.579, 37.21, 186.704, 25, -193.6]
  MoveL 1704 to (33.07, -147.3, 4.06) mm, rotated rx 91.55 ry 0 rz -166.4 deg; joints [122.465, -25.248, 44.541, -117.443, 37.218, 186.555, 25, -193.6]
  MoveL 1705 to (33.05, -147.29, 4.63) mm, rotated rx 91.77 ry 0 rz -166.4 deg; joints [122.509, -25.241, 44.448, -117.304, 37.216, 186.18, 25, -193.597]
  MoveL 1706 to (33.65, -146.86, 10.18) mm, rotated rx 93.75 ry 0 rz -166.15 deg; joints [122.922, -25.146, 43.587, -116.039, 37.221, 182.785, 25, -193.846]
  MoveL 1707 to (33.31, -146.88, 11.08) mm, rotated rx 94.53 ry 0 rz -166.33 deg; joints [123.067, -25.097, 43.282, -115.61, 37.234, 181.515, 25, -193.67]
  MoveL 1708 to (33.12, -146.86, 11.95) mm, rotated rx 94.66 ry 0 rz -166.35 deg; joints [123.107, -25.091, 43.212, -115.5, 37.24, 181.267, 25, -193.654]
  MoveL 1709 to (32.94, -146.65, 14.63) mm, rotated rx 95.61 ry 0 rz -166.39 deg; joints [123.319, -25.021, 42.792, -114.905, 37.273, 179.657, 25, -193.61]
  MoveL 1710 to (31.71, -146.74, 16.44) mm, rotated rx 96.77 ry 0 rz -167.01 deg; joints [123.549, -24.912, 42.31, -114.271, 37.318, 177.781, 25, -192.992]
  MoveL 1711 to (31.44, -146.74, 16.89) mm, rotated rx 96.86 ry 0 rz -167.06 deg; joints [123.577, -24.908, 42.266, -114.2, 37.326, 177.61, 25, -192.938]
  MoveL 1712 to (30.13, -146.72, 19.3) mm, rotated rx 97.78 ry 0 rz -167.55 deg; joints [123.79, -24.818, 41.857, -113.648, 37.382, 176.074, 25, -192.452]
  MoveL 1713 to (29.8, -146.69, 20.02) mm, rotated rx 97.98 ry 0 rz -167.63 deg; joints [123.843, -24.8, 41.764, -113.516, 37.398, 175.727, 25, -192.368]
  MoveL 1714 to (28.15, -146.67, 22.3) mm, rotated rx 99.02 ry 0 rz -168.34 deg; joints [124.076, -24.679, 41.308, -112.932, 37.472, 174.038, 25, -191.658]
  MoveL 1715 to (28.2, -146.65, 22.33) mm, rotated rx 99.35 ry 0 rz -169.54 deg; joints [124.064, -24.508, 41.097, -112.893, 37.446, 173.655, 25, -190.457]
  MoveL 1716 to (24.5, -147.61, 20.46) mm, rotated rx 98.63 ry 0 rz -171 deg; joints [123.892, -24.59, 41.419, -113.315, 37.388, 174.843, 25, -188.998]
  MoveL 1717 to (23.28, -147.84, 20.2) mm, rotated rx 98.63 ry 0 rz -171 deg; joints [123.916, -24.647, 41.465, -113.283, 37.404, 174.81, 25, -188.998]
  MoveL 1718 to (21.71, -148.03, 20.6) mm, rotated rx 98.64 ry 0 rz -171.14 deg; joints [123.953, -24.697, 41.483, -113.216, 37.425, 174.733, 25, -188.858]
  MoveL 1719 to (19.07, -148.15, 22.25) mm, rotated rx 99.27 ry 0 rz -172.15 deg; joints [124.104, -24.625, 41.2, -112.845, 37.476, 173.687, 25, -187.847]
  MoveL 1720 to (17.91, -148.03, 23.97) mm, rotated rx 99.27 ry 0 rz -172.15 deg; joints [124.165, -24.658, 41.17, -112.722, 37.505, 173.554, 25, -187.847]
  MoveL 1721 to (17.88, -147.83, 25.16) mm, rotated rx 99.37 ry 0 rz -172.17 deg; joints [124.206, -24.636, 41.091, -112.622, 37.519, 173.345, 25, -187.832]
  MoveL 1722 to (18.2, -147.53, 26.66) mm, rotated rx 99.95 ry 0 rz -172.03 deg; joints [124.347, -24.564, 40.829, -112.287, 37.572, 172.392, 25, -187.971]
  MoveL 1723 to (18.27, -147.53, 26.58) mm, rotated rx 100.76 ry 0 rz -172.21 deg; joints [124.489, -24.459, 40.531, -111.949, 37.625, 171.21, 25, -187.79]
  MoveL 1724 to (15.91, -147.31, 29.23) mm, rotated rx 101.78 ry 0 rz -173.1 deg; joints [124.744, -24.319, 40.069, -111.374, 37.734, 169.552, 25, -186.897]
  MoveL 1725 to (15.51, -147.25, 29.72) mm, rotated rx 101.84 ry 0 rz -173.16 deg; joints [124.772, -24.316, 40.035, -111.315, 37.748, 169.425, 25, -186.843]
  MoveL 1726 to (14.83, -147.1, 30.8) mm, rotated rx 102.26 ry 0 rz -173.41 deg; joints [124.879, -24.255, 39.845, -111.084, 37.797, 168.749, 25, -186.586]
  MoveL 1727 to (12.15, -147.03, 32.27) mm, rotated rx 103.16 ry 0 rz -174.8 deg; joints [125.07, -24.091, 39.44, -110.66, 37.884, 167.376, 25, -185.205]
  MoveL 1728 to (11.52, -146.98, 32.71) mm, rotated rx 103.25 ry 0 rz -174.91 deg; joints [125.105, -24.088, 39.401, -110.591, 37.903, 167.213, 25, -185.093]
  MoveL 1729 to (9.08, -146.59, 35.18) mm, rotated rx 104.12 ry 0 rz -175.74 deg; joints [125.342, -23.955, 39.002, -110.106, 38.025, 165.805, 25, -184.256]
  MoveL 1730 to (8.71, -146.49, 35.65) mm, rotated rx 104.12 ry 0 rz -175.74 deg; joints [125.361, -23.964, 38.994, -110.073, 38.036, 165.77, 25, -184.256]
  MoveL 1731 to (8.05, -146.3, 36.55) mm, rotated rx 104.57 ry 0 rz -176.06 deg; joints [125.47, -23.885, 38.792, -109.853, 38.093, 165.076, 25, -183.939]
  MoveL 1732 to (8.17, -146.3, 36.55) mm, rotated rx 104.87 ry 0 rz -177.21 deg; joints [125.46, -23.715, 38.597, -109.828, 38.075, 164.74, 25, -182.795]
  MoveL 1733 to (6.9, -146.51, 35.99) mm, rotated rx 104.65 ry 0 rz -177.71 deg; joints [125.402, -23.753, 38.697, -109.943, 38.044, 165.086, 25, -182.293]
  MoveL 1734 to (6.1, -146.6, 35.76) mm, rotated rx 104.62 ry 0 rz -177.85 deg; joints [125.401, -23.779, 38.73, -109.952, 38.045, 165.13, 25, -182.152]
  MoveL 1735 to (1.55, -146.87, 35.12) mm, rotated rx 104.39 ry 0 rz -179.53 deg; joints [125.344, -23.829, 38.845, -110.07, 38.016, 165.494, 25, -180.465]
  MoveL 1736 to (0.94, -146.87, 35.12) mm, rotated rx 104.27 ry 0 rz 179.89 deg; joints [125.3, -23.806, 38.861, -110.146, 37.989, 165.689, 25, -179.885]
  MoveL 1737 to (-2.9, -147.33, 33) mm, rotated rx 103.45 ry 0 rz 178.39 deg; joints [125.085, -23.939, 39.238, -110.588, 37.88, 167.004, 25, -178.393]
  MoveL 1738 to (-3.8, -147.5, 32.22) mm, rotated rx 103.16 ry 0 rz 178.08 deg; joints [125.013, -23.989, 39.372, -110.74, 37.845, 167.454, 25, -178.084]
  MoveL 1739 to (-7.46, -147.74, 30.42) mm, rotated rx 102.47 ry 0 rz 176.67 deg; joints [124.835, -24.094, 39.689, -111.121, 37.76, 168.572, 25, -176.672]
  MoveL 1740 to (-11.67, -148.19, 26.67) mm, rotated rx 100.87 ry 0 rz 174.85 deg; joints [124.429, -24.29, 40.382, -112.018, 37.579, 171.161, 25, -174.846]
  MoveL 1741 to (-12.15, -148.21, 26.31) mm, rotated rx 100.79 ry 0 rz 174.74 deg; joints [124.41, -24.311, 40.43, -112.064, 37.573, 171.291, 25, -174.738]
  MoveL 1742 to (-14.84, -148.24, 24.72) mm, rotated rx 100.23 ry 0 rz 173.79 deg; joints [124.275, -24.393, 40.693, -112.383, 37.521, 172.206, 25, -173.79]
  MoveL 1743 to (-16.01, -148.36, 23.23) mm, rotated rx 99.43 ry 0 rz 173.08 deg; joints [124.076, -24.455, 41.011, -112.844, 37.444, 173.517, 25, -173.084]
  MoveL 1744 to (-16.61, -148.38, 22.69) mm, rotated rx 99.43 ry 0 rz 173.08 deg; joints [124.079, -24.486, 41.048, -112.848, 37.449, 173.524, 25, -173.084]
  MoveL 1745 to (-17.21, -148.37, 22.31) mm, rotated rx 99.29 ry 0 rz 172.86 deg; joints [124.044, -24.503, 41.115, -112.935, 37.436, 173.767, 25, -172.857]
  MoveL 1746 to (-21.4, -148.14, 19.91) mm, rotated rx 98.4 ry 0 rz 171.3 deg; joints [123.835, -24.608, 41.518, -113.457, 37.37, 175.237, 25, -171.302]
  MoveL 1747 to (-21.33, -148.15, 20.01) mm, rotated rx 97.44 ry 0 rz 170.87 deg; joints [123.632, -24.63, 41.813, -113.946, 37.302, 176.732, 25, -170.866]
  MoveL 1748 to (-20.58, -148.81, 15.47) mm, rotated rx 95.71 ry 0 rz 171.19 deg; joints [123.237, -24.785, 42.579, -115, 37.213, 179.642, 25, -171.189]
  MoveL 1749 to (-20.61, -148.91, 14.47) mm, rotated rx 95.71 ry 0 rz 171.19 deg; joints [123.22, -24.793, 42.615, -115.05, 37.21, 179.697, 25, -171.189]
  MoveL 1750 to (-20.84, -148.95, 13.71) mm, rotated rx 95.59 ry 0 rz 171.16 deg; joints [123.19, -24.811, 42.686, -115.137, 37.206, 179.909, 25, -171.163]
  MoveL 1751 to (-21.83, -148.98, 11.55) mm, rotated rx 94.77 ry 0 rz 170.8 deg; joints [123.009, -24.871, 43.046, -115.648, 37.18, 181.304, 25, -170.796]
  MoveL 1752 to (-21.68, -149.16, 9.48) mm, rotated rx 93.52 ry 0 rz 170.78 deg; joints [122.758, -24.931, 43.538, -116.376, 37.155, 183.365, 25, -170.785]
  MoveL 1753 to (-21.88, -149.2, 8.29) mm, rotated rx 93.52 ry 0 rz 170.78 deg; joints [122.743, -24.946, 43.586, -116.429, 37.156, 183.426, 25, -170.785]
  MoveL 1754 to (-22.55, -149.15, 7.3) mm, rotated rx 93.47 ry 0 rz 170.76 deg; joints [122.73, -24.98, 43.657, -116.484, 37.163, 183.545, 25, -170.76]
  MoveL 1755 to (-23.91, -148.99, 6.04) mm, rotated rx 92.99 ry 0 rz 170.24 deg; joints [122.631, -25.004, 43.862, -116.786, 37.16, 184.36, 25, -170.241]
  MoveL 1756 to (-24.53, -148.93, 4.9) mm, rotated rx 92.35 ry 0 rz 169.84 deg; joints [122.499, -25.008, 44.104, -117.181, 37.156, 185.441, 25, -169.836]
  MoveL 1757 to (-24.97, -148.88, 4.36) mm, rotated rx 92.35 ry 0 rz 169.84 deg; joints [122.501, -25.03, 44.135, -117.192, 37.162, 185.455, 25, -169.836]
  MoveL 1758 to (-25.42, -148.81, 3.98) mm, rotated rx 92.29 ry 0 rz 169.76 deg; joints [122.49, -25.046, 44.179, -117.235, 37.166, 185.572, 25, -169.763]
  MoveL 1759 to (-27.35, -148.5, 2.61) mm, rotated rx 91.77 ry 0 rz 169.02 deg; joints [122.385, -25.064, 44.401, -117.567, 37.172, 186.464, 25, -169.02]
  MoveL 1760 to (-29.2, -148.17, 1.12) mm, rotated rx 91.18 ry 0 rz 168.28 deg; joints [122.269, -25.077, 44.645, -117.943, 37.182, 187.473, 25, -168.277]
  MoveL 1761 to (-30.79, -147.85, 0.61) mm, rotated rx 91.18 ry 0 rz 168.28 deg; joints [122.298, -25.153, 44.711, -117.905, 37.201, 187.438, 25, -168.277]
  MoveL 1762 to (-31.85, -147.62, 0.66) mm, rotated rx 91.2 ry 0 rz 167.86 deg; joints [122.301, -25.153, 44.704, -117.894, 37.201, 187.407, 25, -167.864]
  MoveL 1763 to (-33.74, -147.19, 1.72) mm, rotated rx 91.2 ry 0 rz 167.86 deg; joints [122.362, -25.241, 44.727, -117.762, 37.221, 187.268, 25, -167.864]
  MoveL 1764 to (-39.02, -145.58, 9.53) mm, rotated rx 94.16 ry 0 rz 165.77 deg; joints [122.97, -25.11, 43.455, -115.883, 37.22, 182.193, 25, -165.772]
  MoveL 1765 to (-41.85, -144.54, 12.77) mm, rotated rx 95.49 ry 0 rz 164.55 deg; joints [123.251, -25.01, 42.876, -115.077, 37.255, 179.957, 25, -164.552]
  MoveL 1766 to (-42.19, -144.4, 13.29) mm, rotated rx 95.49 ry 0 rz 164.55 deg; joints [123.269, -25.023, 42.869, -115.037, 37.262, 179.913, 25, -164.552]
  MoveL 1767 to (-42.43, -144.28, 13.77) mm, rotated rx 95.68 ry 0 rz 164.45 deg; joints [123.309, -25.009, 42.788, -114.924, 37.269, 179.604, 25, -164.455]
  MoveL 1768 to (-44.48, -143.1, 18.72) mm, rotated rx 97.52 ry 0 rz 163.6 deg; joints [123.731, -24.847, 41.973, -113.799, 37.366, 176.509, 25, -163.604]
  MoveL 1769 to (-47.27, -141.59, 22.89) mm, rotated rx 99.27 ry 0 rz 162.32 deg; joints [124.133, -24.649, 41.197, -112.79, 37.491, 173.628, 25, -162.318]
  MoveL 1770 to (-47.64, -141.33, 23.72) mm, rotated rx 99.43 ry 0 rz 162.25 deg; joints [124.185, -24.637, 41.119, -112.67, 37.511, 173.34, 25, -162.247]
  MoveL 1771 to (-48.96, -140.12, 27.88) mm, rotated rx 100.98 ry 0 rz 161.64 deg; joints [124.569, -24.441, 40.417, -111.774, 37.661, 170.796, 25, -161.641]
  MoveL 1772 to (-49.1, -139.98, 28.33) mm, rotated rx 101.16 ry 0 rz 161.57 deg; joints [124.614, -24.416, 40.335, -111.672, 37.68, 170.5, 25, -161.568]
  MoveL 1773 to (-50.03, -138.68, 32.76) mm, rotated rx 102.79 ry 0 rz 161.1 deg; joints [125.032, -24.179, 39.589, -110.758, 37.871, 167.86, 25, -161.099]
  MoveL 1774 to (-50.07, -138.48, 33.54) mm, rotated rx 102.88 ry 0 rz 161.09 deg; joints [125.07, -24.162, 39.53, -110.681, 37.89, 167.685, 25, -161.095]
  MoveL 1775 to (-50.26, -138.3, 33.93) mm, rotated rx 103.36 ry 0 rz 160.92 deg; joints [125.172, -24.088, 39.334, -110.464, 37.94, 166.958, 25, -160.92]
  MoveL 1776 to (-50.22, -138.32, 33.9) mm, rotated rx 103.85 ry 0 rz 159.68 deg; joints [125.195, -23.889, 39.066, -110.365, 37.937, 166.351, 25, -159.68]
  MoveL 1777 to (-52.26, -137.77, 33.08) mm, rotated rx 103.53 ry 0 rz 158.86 deg; joints [125.111, -23.941, 39.213, -110.537, 37.894, 166.861, 25, -158.865]
  MoveL 1778 to (-53.42, -137.37, 32.92) mm, rotated rx 103.53 ry 0 rz 158.86 deg; joints [125.137, -23.995, 39.254, -110.504, 37.913, 166.827, 25, -158.865]
  MoveL 1779 to (-54.01, -137.12, 33) mm, rotated rx 103.56 ry 0 rz 158.62 deg; joints [125.144, -23.991, 39.241, -110.488, 37.916, 166.781, 25, -158.615]
  MoveL 1780 to (-55.34, -136.41, 33.71) mm, rotated rx 103.56 ry 0 rz 158.62 deg; joints [125.195, -24.045, 39.257, -110.406, 37.949, 166.695, 25, -158.615]
  MoveL 1781 to (-59.26, -133.49, 38.41) mm, rotated rx 105.4 ry 0 rz 156.77 deg; joints [125.679, -23.735, 38.415, -109.44, 38.207, 163.791, 25, -156.766]
  MoveL 1782 to (-59.52, -133.29, 38.71) mm, rotated rx 105.54 ry 0 rz 156.62 deg; joints [125.713, -23.709, 38.352, -109.373, 38.226, 163.578, 25, -156.619]
  MoveL 1783 to (-64.29, -130.15, 41.64) mm, rotated rx 106.83 ry 0 rz 154.19 deg; joints [126.042, -23.454, 37.752, -108.748, 38.415, 161.586, 25, -154.193]
  MoveL 1784 to (-64.9, -129.68, 42.18) mm, rotated rx 106.96 ry 0 rz 154.04 deg; joints [126.089, -23.442, 37.697, -108.666, 38.444, 161.376, 25, -154.039]
  MoveL 1785 to (-67.67, -127.47, 44.47) mm, rotated rx 108.06 ry 0 rz 151.89 deg; joints [126.334, -23.151, 37.148, -108.204, 38.588, 159.752, 25, -151.886]
  MoveL 1786 to (-68.58, -127.04, 44.33) mm, rotated rx 108.01 ry 0 rz 151.48 deg; joints [126.318, -23.163, 37.176, -108.232, 38.577, 159.843, 25, -151.484]
  MoveL 1787 to (-69.23, -126.7, 44.28) mm, rotated rx 108 ry 0 rz 151.3 deg; joints [126.321, -23.176, 37.188, -108.229, 38.58, 159.849, 25, -151.3]
  MoveL 1788 to (-73.83, -124.07, 44.3) mm, rotated rx 108.01 ry 0 rz 149.25 deg; joints [126.327, -23.18, 37.188, -108.221, 38.584, 159.832, 25, -149.249]
  MoveL 1789 to (-74.21, -123.86, 44.26) mm, rotated rx 107.99 ry 0 rz 149 deg; joints [126.317, -23.176, 37.19, -108.236, 38.578, 159.865, 25, -149]
  MoveL 1790 to (-79.86, -120.38, 44.03) mm, rotated rx 107.9 ry 0 rz 146.41 deg; joints [126.295, -23.197, 37.234, -108.276, 38.564, 159.998, 25, -146.406]
  MoveL 1791 to (-80.54, -119.9, 44.09) mm, rotated rx 107.92 ry 0 rz 146.2 deg; joints [126.308, -23.207, 37.235, -108.257, 38.573, 159.959, 25, -146.202]
  MoveL 1792 to (-84.53, -116.94, 44.58) mm, rotated rx 108.11 ry 0 rz 144.24 deg; joints [126.362, -23.169, 37.145, -108.162, 38.607, 159.66, 25, -144.239]
  Set speed (16.7 mm/s)
  MoveL 1793 to (-95.84, -132.21, 50.82) mm, rotated rx 108.12 ry 0 rz 144.14 deg; joints [125.883, -23.688, 37.004, -107.661, 37.961, 158.87, 25, -144.142]
  Set speed (1000.0 mm/s)
  MoveL 1794 to (-98.33, -130.06, 51.52) mm, rotated rx 108.35 ry 0 rz 143.13 deg; joints [125.96, -23.655, 36.905, -107.533, 38.013, 158.504, 25, -143.132]
  Set speed (5.0 mm/s)
  MoveL 1795 to (-86.94, -114.87, 45.23) mm, rotated rx 108.35 ry 0 rz 143.13 deg; joints [126.439, -23.135, 37.045, -108.035, 38.657, 159.286, 25, -143.132]
  Set speed (16.7 mm/s)
  MoveL 1796 to (-87.73, -114.16, 45.49) mm, rotated rx 108.45 ry 0 rz 142.71 deg; joints [126.468, -23.114, 36.996, -107.984, 38.675, 159.125, 25, -142.713]
  Set speed (16.7 mm/s)
  MoveL 1797 to (-99.22, -129.26, 51.82) mm, rotated rx 108.45 ry 0 rz 142.71 deg; joints [125.991, -23.633, 36.855, -107.481, 38.032, 158.341, 25, -142.713]
  Set speed (1000.0 mm/s)
  MoveL 1798 to (-108.79, -120.03, 54.78) mm, rotated rx 109.49 ry 0 rz 138.04 deg; joints [126.293, -23.407, 36.358, -106.971, 38.233, 156.737, 25, -138.038]
  Set speed (5.0 mm/s)
  MoveL 1799 to (-96.18, -106.01, 48.11) mm, rotated rx 109.49 ry 0 rz 138.04 deg; joints [126.758, -22.897, 36.512, -107.492, 38.862, 157.54, 25, -138.038]
  Set speed (16.7 mm/s)
  MoveL 1800 to (-99.42, -102.43, 49.31) mm, rotated rx 109.98 ry 0 rz 136.11 deg; joints [126.893, -22.794, 36.288, -107.269, 38.951, 156.813, 25, -136.113]
  MoveL 1801 to (-100.01, -101.64, 49.73) mm, rotated rx 110.06 ry 0 rz 135.94 deg; joints [126.936, -22.793, 36.254, -107.204, 38.981, 156.654, 25, -135.936]
  MoveL 1802 to (-101.98, -98.93, 51.18) mm, rotated rx 110.67 ry 0 rz 134.56 deg; joints [127.102, -22.656, 35.972, -106.936, 39.093, 155.755, 25, -134.557]
  MoveL 1803 to (-102.57, -97.95, 51.87) mm, rotated rx 110.86 ry 0 rz 134.27 deg; joints [127.172, -22.625, 35.885, -106.83, 39.142, 155.446, 25, -134.271]
  MoveL 1804 to (-104.87, -93.14, 55.92) mm, rotated rx 112.45 ry 0 rz 132.28 deg; joints [127.636, -22.26, 35.142, -106.125, 39.468, 153.078, 25, -132.277]
  MoveL 1805 to (-104.81, -93.16, 56.04) mm, rotated rx 111.29 ry 0 rz 130.76 deg; joints [127.283, -22.322, 35.46, -106.623, 39.211, 154.787, 25, -130.764]
  MoveL 1806 to (-104.67, -93.92, 55.05) mm, rotated rx 110.88 ry 0 rz 131.03 deg; joints [127.167, -22.415, 35.649, -106.803, 39.13, 155.39, 25, -131.035]
  MoveL 1807 to (-104.54, -94.17, 54.86) mm, rotated rx 110.64 ry 0 rz 131.28 deg; joints [127.117, -22.474, 35.754, -106.885, 39.097, 155.719, 25, -131.28]
  MoveL 1808 to (-102.34, -98.93, 50.44) mm, rotated rx 108.57 ry 0 rz 133.99 deg; joints [126.591, -22.979, 36.738, -107.763, 38.751, 158.766, 25, -133.99]
  MoveL 1809 to (-101.03, -100.32, 50.38) mm, rotated rx 108.54 ry 0 rz 134.76 deg; joints [126.583, -22.985, 36.751, -107.776, 38.746, 158.808, 25, -134.76]
  MoveL 1810 to (-100.46, -100.97, 50.2) mm, rotated rx 108.54 ry 0 rz 134.76 deg; joints [126.558, -22.953, 36.734, -107.809, 38.728, 158.843, 25, -134.76]
  MoveL 1811 to (-99.81, -102.26, 48.86) mm, rotated rx 108.54 ry 0 rz 134.76 deg; joints [126.494, -22.92, 36.748, -107.904, 38.682, 158.945, 25, -134.76]
  MoveL 1812 to (-99.79, -102.49, 48.42) mm, rotated rx 108.38 ry 0 rz 134.82 deg; joints [126.448, -22.952, 36.822, -107.982, 38.653, 159.188, 25, -134.824]
  MoveL 1813 to (-99.7, -103.53, 46.31) mm, rotated rx 107.54 ry 0 rz 135.14 deg; joints [126.217, -23.12, 37.211, -108.389, 38.509, 160.476, 25, -135.141]
  MoveL 1814 to (-99.77, -103.45, 46.33) mm, rotated rx 107 ry 0 rz 136.45 deg; joints [126.182, -23.344, 37.502, -108.492, 38.499, 161.135, 25, -136.447]
  MoveL 1815 to (-96.16, -106, 48.23) mm, rotated rx 107.76 ry 0 rz 138.2 deg; joints [126.39, -23.194, 37.152, -108.122, 38.627, 159.97, 25, -138.2]
  Set speed (16.7 mm/s)
  MoveL 1816 to (-108.85, -120.19, 54.33) mm, rotated rx 107.76 ry 0 rz 138.2 deg; joints [125.907, -23.718, 37.02, -107.629, 37.978, 159.196, 25, -138.2]
  Set speed (1000.0 mm/s)
  MoveL 1817 to (-95.78, -132.54, 50.07) mm, rotated rx 106.41 ry 0 rz 143.55 deg; joints [125.447, -23.885, 37.602, -108.423, 37.682, 161.416, 25, -143.552]
  Set speed (5.0 mm/s)
  MoveL 1818 to (-84.39, -117.1, 44.42) mm, rotated rx 106.41 ry 0 rz 143.55 deg; joints [125.945, -23.351, 37.716, -108.889, 38.347, 162.161, 25, -143.552]
  Set speed (16.7 mm/s)
  MoveL 1819 to (-81.74, -120.21, 40.92) mm, rotated rx 105.02 ry 0 rz 145.12 deg; joints [125.573, -23.603, 38.354, -109.595, 38.134, 164.327, 25, -145.121]
  MoveL 1820 to (-81.42, -121.13, 38.81) mm, rotated rx 105.02 ry 0 rz 145.12 deg; joints [125.507, -23.601, 38.413, -109.713, 38.095, 164.455, 25, -145.121]
  MoveL 1821 to (-82.02, -121.15, 37.44) mm, rotated rx 104.91 ry 0 rz 145.1 deg; joints [125.464, -23.655, 38.519, -109.806, 38.073, 164.674, 25, -145.105]
  MoveL 1822 to (-84.98, -120.27, 33.5) mm, rotated rx 103.37 ry 0 rz 143.97 deg; joints [125.062, -23.908, 39.223, -110.623, 37.864, 167.113, 25, -143.968]
  MoveL 1823 to (-85.5, -120.05, 32.94) mm, rotated rx 103.3 ry 0 rz 143.88 deg; joints [125.043, -23.939, 39.281, -110.669, 37.856, 167.24, 25, -143.884]
  MoveL 1824 to (-86.68, -119.46, 31.98) mm, rotated rx 102.39 ry 0 rz 143.08 deg; joints [124.82, -24.027, 39.621, -111.131, 37.746, 168.661, 25, -143.08]
  MoveL 1825 to (-86.92, -119.52, 31.09) mm, rotated rx 102.04 ry 0 rz 143.02 deg; joints [124.732, -24.078, 39.778, -111.322, 37.706, 169.216, 25, -143.019]
  MoveL 1826 to (-87.44, -119.42, 30.02) mm, rotated rx 102.04 ry 0 rz 143.02 deg; joints [124.721, -24.111, 39.832, -111.355, 37.703, 169.254, 25, -143.019]
  MoveL 1827 to (-88.11, -119.1, 29.31) mm, rotated rx 101.98 ry 0 rz 142.97 deg; joints [124.707, -24.153, 39.899, -111.396, 37.7, 169.367, 25, -142.968]
  MoveL 1828 to (-90.45, -117.76, 27.55) mm, rotated rx 101.3 ry 0 rz 141.94 deg; joints [124.537, -24.248, 40.207, -111.777, 37.626, 170.469, 25, -141.935]
  MoveL 1829 to (-90.79, -117.56, 27.27) mm, rotated rx 101.22 ry 0 rz 141.82 deg; joints [124.518, -24.264, 40.249, -111.821, 37.619, 170.598, 25, -141.823]
  MoveL 1830 to (-93.09, -116.11, 25.68) mm, rotated rx 100.61 ry 0 rz 140.79 deg; joints [124.366, -24.346, 40.526, -112.17, 37.557, 171.598, 25, -140.785]
  MoveL 1831 to (-95.54, -114.51, 23.8) mm, rotated rx 99.86 ry 0 rz 139.63 deg; joints [124.182, -24.435, 40.857, -112.601, 37.486, 172.823, 25, -139.635]
  MoveL 1832 to (-96.15, -114.07, 23.47) mm, rotated rx 99.86 ry 0 rz 139.63 deg; joints [124.193, -24.472, 40.892, -112.589, 37.495, 172.813, 25, -139.635]
  MoveL 1833 to (-96.7, -113.64, 23.29) mm, rotated rx 99.79 ry 0 rz 139.37 deg; joints [124.177, -24.48, 40.922, -112.629, 37.489, 172.924, 25, -139.366]
  MoveL 1834 to (-100.85, -110.19, 22.17) mm, rotated rx 99.37 ry 0 rz 137.34 deg; joints [124.078, -24.535, 41.115, -112.871, 37.454, 173.615, 25, -137.339]
  MoveL 1835 to (-102.57, -109.05, 19.9) mm, rotated rx 98.21 ry 0 rz 136.05 deg; joints [123.785, -24.598, 41.567, -113.568, 37.35, 175.546, 25, -136.047]
  MoveL 1836 to (-103.23, -108.52, 19.3) mm, rotated rx 98.21 ry 0 rz 136.05 deg; joints [123.793, -24.64, 41.614, -113.566, 37.359, 175.547, 25, -136.047]
  MoveL 1837 to (-103.63, -108.19, 19.07) mm, rotated rx 98.12 ry 0 rz 135.85 deg; joints [123.773, -24.649, 41.652, -113.617, 37.353, 175.69, 25, -135.849]
  MoveL 1838 to (-108.47, -103.62, 17.48) mm, rotated rx 97.57 ry 0 rz 133.47 deg; joints [123.651, -24.726, 41.916, -113.94, 37.322, 176.604, 25, -133.472]
  MoveL 1839 to (-110.72, -101.49, 15.76) mm, rotated rx 96.83 ry 0 rz 132.05 deg; joints [123.47, -24.766, 42.219, -114.401, 37.272, 177.861, 25, -132.053]
  MoveL 1840 to (-111.18, -101.03, 15.52) mm, rotated rx 96.83 ry 0 rz 132.05 deg; joints [123.48, -24.797, 42.247, -114.389, 37.28, 177.85, 25, -132.053]
  MoveL 1841 to (-111.55, -100.62, 15.43) mm, rotated rx 96.81 ry 0 rz 131.99 deg; joints [123.485, -24.816, 42.266, -114.386, 37.284, 177.861, 25, -131.99]
  MoveL 1842 to (-112.64, -99.43, 15.33) mm, rotated rx 96.77 ry 0 rz 131.37 deg; joints [123.476, -24.819, 42.284, -114.41, 37.282, 177.928, 25, -131.374]
  MoveL 1843 to (-114.5, -97.43, 14.34) mm, rotated rx 96.35 ry 0 rz 130.09 deg; joints [123.367, -24.826, 42.447, -114.687, 37.253, 178.659, 25, -130.087]
  MoveL 1844 to (-114.93, -96.94, 14.2) mm, rotated rx 96.33 ry 0 rz 129.99 deg; joints [123.371, -24.845, 42.47, -114.688, 37.257, 178.679, 25, -129.986]
  MoveL 1845 to (-116.59, -94.97, 13.94) mm, rotated rx 96.24 ry 0 rz 129.07 deg; joints [123.354, -24.861, 42.515, -114.737, 37.255, 178.825, 25, -129.071]
  MoveL 1846 to (-116.84, -94.68, 13.79) mm, rotated rx 96.15 ry 0 rz 128.76 deg; joints [123.326, -24.848, 42.538, -114.803, 37.245, 178.984, 25, -128.76]
  MoveL 1847 to (-120.24, -90.43, 12.79) mm, rotated rx 95.79 ry 0 rz 126.78 deg; joints [123.251, -24.887, 42.705, -115.019, 37.234, 179.587, 25, -126.776]
  Set speed (16.7 mm/s)
  MoveL 1848 to (-136.18, -102.35, 14.8) mm, rotated rx 95.79 ry 0 rz 126.78 deg; joints [122.64, -25.494, 42.731, -114.826, 36.462, 179.117, 25, -126.776]
  Set speed (1000.0 mm/s)
  MoveL 1849 to (-140.14, -95.07, 23.87) mm, rotated rx 98.56 ry 0 rz 124.8 deg; joints [123.373, -25.318, 41.508, -112.942, 36.68, 174.266, 25, -124.803]
  Set speed (5.0 mm/s)
  MoveL 1850 to (-123.9, -83.78, 20.89) mm, rotated rx 98.56 ry 0 rz 124.8 deg; joints [123.957, -24.727, 41.519, -113.22, 37.431, 174.822, 25, -124.803]
  Set speed (16.7 mm/s)
  MoveL 1851 to (-124.07, -83.45, 21.18) mm, rotated rx 98.78 ry 0 rz 124.55 deg; joints [123.998, -24.692, 41.422, -113.113, 37.442, 174.479, 25, -124.553]
  MoveL 1852 to (-124.96, -81.65, 22.89) mm, rotated rx 99.43 ry 0 rz 123.79 deg; joints [124.154, -24.617, 41.13, -112.731, 37.495, 173.403, 25, -123.791]
  MoveL 1853 to (-125.25, -80.96, 23.76) mm, rotated rx 99.82 ry 0 rz 123.75 deg; joints [124.261, -24.598, 40.977, -112.489, 37.539, 172.744, 25, -123.749]
  MoveL 1854 to (-124.73, -80.95, 26.31) mm, rotated rx 100.71 ry 0 rz 123.65 deg; joints [124.472, -24.46, 40.552, -111.986, 37.618, 171.293, 25, -123.655]
  MoveL 1855 to (-125.37, -79.47, 27.83) mm, rotated rx 101.3 ry 0 rz 123.04 deg; joints [124.617, -24.381, 40.288, -111.655, 37.678, 170.342, 25, -123.045]
  MoveL 1856 to (-125.5, -79.1, 28.27) mm, rotated rx 101.37 ry 0 rz 122.99 deg; joints [124.646, -24.378, 40.251, -111.594, 37.692, 170.2, 25, -122.986]
  MoveL 1857 to (-125.87, -77.67, 30.51) mm, rotated rx 102.15 ry 0 rz 122.5 deg; joints [124.85, -24.271, 39.895, -111.145, 37.784, 168.926, 25, -122.502]
  MoveL 1858 to (-126.01, -77.35, 30.76) mm, rotated rx 102.41 ry 0 rz 122.24 deg; joints [124.9, -24.223, 39.78, -111.03, 37.805, 168.534, 25, -122.238]
  MoveL 1859 to (-128.01, -71.29, 36.59) mm, rotated rx 104.7 ry 0 rz 119.79 deg; joints [125.492, -23.854, 38.734, -109.804, 38.104, 164.885, 25, -119.794]
  MoveL 1860 to (-128.08, -70.51, 37.83) mm, rotated rx 104.7 ry 0 rz 119.79 deg; joints [125.537, -23.867, 38.706, -109.727, 38.131, 164.801, 25, -119.794]
  MoveL 1861 to (-127.99, -70.35, 38.41) mm, rotated rx 104.8 ry 0 rz 119.77 deg; joints [125.57, -23.848, 38.652, -109.662, 38.149, 164.638, 25, -119.774]
  MoveL 1862 to (-127.73, -70.1, 39.72) mm, rotated rx 105.31 ry 0 rz 119.74 deg; joints [125.707, -23.757, 38.416, -109.396, 38.225, 163.83, 25, -119.74]
  MoveL 1863 to (-127.97, -68.59, 41.54) mm, rotated rx 106.53 ry 0 rz 118.98 deg; joints [125.994, -23.533, 37.889, -108.846, 38.389, 162.001, 25, -118.984]
  MoveL 1864 to (-128.66, -66.29, 43.13) mm, rotated rx 107.37 ry 0 rz 117.83 deg; joints [126.196, -23.358, 37.507, -108.471, 38.508, 160.749, 25, -117.831]
  MoveL 1865 to (-128.78, -65.7, 43.67) mm, rotated rx 107.37 ry 0 rz 117.83 deg; joints [126.223, -23.373, 37.502, -108.431, 38.526, 160.706, 25, -117.831]
  MoveL 1866 to (-128.8, -65.27, 44.25) mm, rotated rx 107.44 ry 0 rz 117.78 deg; joints [126.258, -23.363, 37.46, -108.371, 38.549, 160.569, 25, -117.776]
  MoveL 1867 to (-128.69, -64.22, 46.08) mm, rotated rx 108.17 ry 0 rz 117.42 deg; joints [126.458, -23.218, 37.123, -108.018, 38.673, 159.453, 25, -117.424]
  MoveL 1868 to (-128.72, -63.87, 46.47) mm, rotated rx 108.46 ry 0 rz 117.21 deg; joints [126.526, -23.155, 36.995, -107.899, 38.716, 159.027, 25, -117.213]
  MoveL 1869 to (-129.16, -61.26, 48.69) mm, rotated rx 109.5 ry 0 rz 116.07 deg; joints [126.798, -22.931, 36.519, -107.436, 38.891, 157.479, 25, -116.068]
  MoveL 1870 to (-129.09, -61.41, 48.69) mm, rotated rx 108.26 ry 0 rz 114.62 deg; joints [126.436, -22.98, 36.865, -108.007, 38.647, 159.338, 25, -114.623]
  MoveL 1871 to (-128.97, -64.41, 44.99) mm, rotated rx 106.78 ry 0 rz 115.73 deg; joints [126.03, -23.272, 37.549, -108.729, 38.396, 161.612, 25, -115.731]
  MoveL 1872 to (-128.99, -64.74, 44.48) mm, rotated rx 106.78 ry 0 rz 115.73 deg; joints [126.011, -23.268, 37.56, -108.76, 38.384, 161.646, 25, -115.731]
  MoveL 1873 to (-129.25, -65.47, 42.6) mm, rotated rx 106.16 ry 0 rz 115.9 deg; joints [125.833, -23.386, 37.856, -109.088, 38.279, 162.63, 25, -115.903]
  MoveL 1874 to (-129.24, -65.64, 42.38) mm, rotated rx 105.8 ry 0 rz 116.09 deg; joints [125.759, -23.454, 38.004, -109.232, 38.237, 163.15, 25, -116.088]
  MoveL 1875 to (-128.22, -70.09, 38.13) mm, rotated rx 103.96 ry 0 rz 117.97 deg; joints [125.288, -23.782, 38.843, -110.161, 37.98, 166.018, 25, -117.966]
  MoveL 1876 to (-128.17, -70.82, 36.94) mm, rotated rx 103.96 ry 0 rz 117.97 deg; joints [125.246, -23.77, 38.87, -110.236, 37.956, 166.099, 25, -117.966]
  MoveL 1877 to (-128.22, -70.97, 36.46) mm, rotated rx 103.77 ry 0 rz 118.01 deg; joints [125.197, -23.801, 38.957, -110.337, 37.93, 166.401, 25, -118.009]
  MoveL 1878 to (-128.78, -71.68, 32.9) mm, rotated rx 101.85 ry 0 rz 118.49 deg; joints [124.752, -24.117, 39.807, -111.295, 37.72, 169.386, 25, -118.491]
  MoveL 1879 to (-127.36, -75.53, 29.71) mm, rotated rx 100.61 ry 0 rz 120.07 deg; joints [124.441, -24.29, 40.368, -111.991, 37.585, 171.398, 25, -120.066]
  MoveL 1880 to (-127.19, -76.01, 29.19) mm, rotated rx 100.61 ry 0 rz 120.07 deg; joints [124.419, -24.274, 40.373, -112.033, 37.573, 171.443, 25, -120.066]
  MoveL 1881 to (-127.12, -76.28, 28.8) mm, rotated rx 100.45 ry 0 rz 120.17 deg; joints [124.382, -24.294, 40.442, -112.12, 37.558, 171.693, 25, -120.174]
  MoveL 1882 to (-127.06, -76.58, 28.26) mm, rotated rx 100.45 ry 0 rz 120.17 deg; joints [124.364, -24.288, 40.454, -112.155, 37.549, 171.731, 25, -120.174]
  MoveL 1883 to (-126.91, -77.99, 24.86) mm, rotated rx 99.14 ry 0 rz 120.67 deg; joints [124.044, -24.449, 41.044, -112.914, 37.43, 173.885, 25, -120.672]
  MoveL 1884 to (-124.48, -82.65, 21.91) mm, rotated rx 97.52 ry 0 rz 123.11 deg; joints [123.71, -24.665, 41.754, -113.772, 37.333, 176.467, 25, -123.113]
  MoveL 1885 to (-124.18, -83.21, 21.54) mm, rotated rx 97.39 ry 0 rz 123.33 deg; joints [123.678, -24.675, 41.812, -113.854, 37.323, 176.689, 25, -123.331]
  Set speed (16.7 mm/s)
  MoveL 1886 to (-140.53, -94.5, 23.78) mm, rotated rx 97.34 ry 0 rz 123.38 deg; joints [123.063, -25.265, 41.834, -113.658, 36.557, 176.263, 25, -123.383]
  Set speed (1000.0 mm/s)
  MoveL 1887 to (-136.26, -102.31, 14.35) mm, rotated rx 94.11 ry 0 rz 126.44 deg; joints [122.318, -25.553, 43.298, -115.724, 36.401, 181.792, 25, -126.439]
  Set speed (5.0 mm/s)
  MoveL 1888 to (-120.21, -90.46, 12.91) mm, rotated rx 94.11 ry 0 rz 126.44 deg; joints [122.943, -24.938, 43.25, -115.867, 37.182, 182.212, 25, -126.439]
  Set speed (16.7 mm/s)
  MoveL 1889 to (-119.01, -92.24, 11.51) mm, rotated rx 93.58 ry 0 rz 127.25 deg; joints [122.828, -24.971, 43.482, -116.203, 37.172, 183.122, 25, -127.255]
  MoveL 1890 to (-118.99, -92.27, 11.51) mm, rotated rx 93.45 ry 0 rz 128.03 deg; joints [122.853, -25.068, 43.585, -116.188, 37.196, 183.239, 25, -128.03]
  MoveL 1891 to (-117.48, -94.12, 12.12) mm, rotated rx 93.68 ry 0 rz 128.94 deg; joints [122.902, -25.055, 43.484, -116.042, 37.199, 182.843, 25, -128.935]
  MoveL 1892 to (-117.07, -94.62, 12.21) mm, rotated rx 93.69 ry 0 rz 129.02 deg; joints [122.895, -25.035, 43.466, -116.051, 37.194, 182.845, 25, -129.018]
  MoveL 1893 to (-115.83, -96.13, 12.2) mm, rotated rx 93.68 ry 0 rz 129.68 deg; joints [122.888, -25.025, 43.462, -116.063, 37.191, 182.863, 25, -129.68]
  MoveL 1894 to (-114.39, -97.74, 13.03) mm, rotated rx 94.06 ry 0 rz 130.83 deg; joints [122.985, -25.043, 43.332, -115.804, 37.209, 182.205, 25, -130.834]
  MoveL 1895 to (-113.7, -98.51, 13.23) mm, rotated rx 94.09 ry 0 rz 131.04 deg; joints [122.983, -25.018, 43.3, -115.798, 37.204, 182.166, 25, -131.044]
  MoveL 1896 to (-109.74, -102.86, 13.59) mm, rotated rx 94.22 ry 0 rz 133.2 deg; joints [123.006, -25, 43.237, -115.724, 37.204, 181.953, 25, -133.202]
  MoveL 1897 to (-109.47, -103.13, 13.66) mm, rotated rx 94.25 ry 0 rz 133.44 deg; joints [123.02, -25.008, 43.228, -115.692, 37.208, 181.88, 25, -133.442]
  MoveL 1898 to (-106.27, -106.28, 14.78) mm, rotated rx 94.69 ry 0 rz 135.23 deg; joints [123.119, -24.988, 43.044, -115.412, 37.223, 181.128, 25, -135.234]
  MoveL 1899 to (-105.7, -106.84, 14.84) mm, rotated rx 94.69 ry 0 rz 135.23 deg; joints [123.102, -24.951, 43.018, -115.44, 37.212, 181.155, 25, -135.234]
  MoveL 1900 to (-104.6, -108.02, 14.08) mm, rotated rx 94.69 ry 0 rz 135.23 deg; joints [123.051, -24.883, 42.997, -115.54, 37.19, 181.261, 25, -135.234]
  MoveL 1901 to (-104.3, -108.37, 13.6) mm, rotated rx 94.51 ry 0 rz 135.41 deg; joints [123.012, -24.895, 43.076, -115.653, 37.184, 181.57, 25, -135.408]
  MoveL 1902 to (-103.93, -108.96, 11.62) mm, rotated rx 94.51 ry 0 rz 135.41 deg; joints [122.962, -24.875, 43.126, -115.779, 37.172, 181.708, 25, -135.408]
  MoveL 1903 to (-104.45, -108.84, 7.2) mm, rotated rx 92.83 ry 0 rz 135.23 deg; joints [122.607, -24.968, 43.852, -116.837, 37.151, 184.574, 25, -135.234]
  MoveL 1904 to (-104.58, -108.76, 6.57) mm, rotated rx 92.77 ry 0 rz 135.22 deg; joints [122.588, -24.977, 43.898, -116.896, 37.152, 184.703, 25, -135.216]
  MoveL 1905 to (-104.79, -108.62, 5.38) mm, rotated rx 92.25 ry 0 rz 135.1 deg; joints [122.483, -24.996, 44.114, -117.222, 37.153, 185.594, 25, -135.101]
  MoveL 1906 to (-105.18, -108.3, 4.15) mm, rotated rx 91.97 ry 0 rz 134.97 deg; joints [122.423, -25.015, 44.255, -117.419, 37.158, 186.093, 25, -134.973]
  MoveL 1907 to (-108.36, -105.17, -2.01) mm, rotated rx 89.8 ry 0 rz 133.38 deg; joints [122.001, -25.076, 45.193, -118.829, 37.222, 189.855, 25, -133.378]
  MoveL 1908 to (-108.65, -104.83, -3.64) mm, rotated rx 88.89 ry 0 rz 133.07 deg; joints [121.836, -25.06, 45.533, -119.393, 37.259, 191.398, 25, -133.068]
  MoveL 1909 to (-108.84, -104.61, -4.29) mm, rotated rx 88.89 ry 0 rz 133.07 deg; joints [121.833, -25.074, 45.564, -119.415, 37.265, 191.424, 25, -133.068]
